LIN {X 0,Y 530.55,Z 455.718,A -85,B 0,C 180,E1 -4236.847,E2 -4236.847} C_VEL
LIN {X 0,Y 530.637,Z 451.254,A -85,B 0,C 180,E1 -4237.994,E2 -4237.994} C_VEL
LIN {X 0,Y 530.743,Z 445.924,A -85,B 0,C 180,E1 -4239.143,E2 -4239.143} C_VEL
LIN {X 0,Y 530.926,Z 439.642,A -85,B 0,C 180,E1 -4240.294,E2 -4240.294} C_VEL
LIN {X 0,Y 531.066,Z 432.27,A -85,B 0,C 180,E1 -4241.449,E2 -4241.449} C_VEL
LIN {X 0,Y 531.288,Z 425.199,A -85,B 0,C 180,E1 -4242.413,E2 -4242.413} C_VEL
LIN {X 0,Y 531.562,Z 417.094,A -85,B 0,C 180,E1 -4243.378,E2 -4243.378} C_VEL
LIN {X 0,Y 531.915,Z 406.759,A -85,B 0,C 180,E1 -4244.441,E2 -4244.441} C_VEL
LIN {X 0,Y 532.284,Z 397.021,A -85,B 0,C 180,E1 -4245.312,E2 -4245.312} C_VEL
LIN {X 0,Y 532.714,Z 385.569,A -85,B 0,C 180,E1 -4246.182,E2 -4246.182} C_VEL
LIN {X 0,Y 533.174,Z 371.646,A -85,B 0,C 180,E1 -4247.055,E2 -4247.055} C_VEL
LIN {X 0,Y 533.562,Z 358.553,A -85,B 0,C 180,E1 -4247.709,E2 -4247.709} C_VEL
LIN {X 0,Y 533.92,Z 343.815,A -85,B 0,C 180,E1 -4248.282,E2 -4248.282} C_VEL
LIN {X 0,Y 534.06,Z 328.911,A -85,B 0,C 180,E1 -4248.704,E2 -4248.704} C_VEL
LIN {X 0,Y 530.589,Z 315.52,A -85,B 0,C 180,E1 -4249.112,E2 -4249.112} C_VEL
LIN {X 0,Y 530.644,Z 311.471,A -85,B 0,C 180,E1 -4252.013,E2 -4252.013} C_VEL
LIN {X 0,Y 530.676,Z 307.059,A -85,B 0,C 180,E1 -4255.074,E2 -4255.074} C_VEL
LIN {X 0,Y 530.747,Z 303.383,A -85,B 0,C 180,E1 -4257.61,E2 -4257.61} C_VEL
LIN {X 0,Y 530.763,Z 299.76,A -85,B 0,C 180,E1 -4260.21,E2 -4260.21} C_VEL
LIN {X 0,Y 530.839,Z 296.13,A -85,B 0,C 180,E1 -4262.875,E2 -4262.875} C_VEL
LIN {X 0,Y 530.854,Z 292.306,A -85,B 0,C 180,E1 -4265.628,E2 -4265.628} C_VEL
LIN {X 0,Y 530.927,Z 287.779,A -85,B 0,C 180,E1 -4268.648,E2 -4268.648} C_VEL
LIN {X 0,Y 530.86,Z 284.993,A -85,B 0,C 180,E1 -4270.444,E2 -4270.444} C_VEL
LIN {X 0,Y 530.946,Z 284.975,A -85,B 0,C 180,E1 -4273.279,E2 -4273.279} C_VEL
LIN {X 0,Y 530.982,Z 284.971,A -85,B 0,C 180,E1 -4275.621,E2 -4275.621} C_VEL
LIN {X 0,Y 530.994,Z 284.97,A -85,B 0,C 180,E1 -4278.564,E2 -4278.564} C_VEL
LIN {X 0,Y 530.95,Z 284.971,A -85,B 0,C 180,E1 -4281.529,E2 -4281.529} C_VEL
LIN {X 0,Y 530.959,Z 284.97,A -85,B 0,C 180,E1 -4284.38,E2 -4284.38} C_VEL
LIN {X 0,Y 530.968,Z 284.973,A -85,B 0,C 180,E1 -4287.133,E2 -4287.133} C_VEL
LIN {X 0,Y 530.95,Z 284.97,A -85,B 0,C 180,E1 -4289.802,E2 -4289.802} C_VEL
LIN {X 0,Y 530.954,Z 284.97,A -85,B 0,C 180,E1 -4292.48,E2 -4292.48} C_VEL
LIN {X 0,Y 530.979,Z 284.967,A -85,B 0,C 180,E1 -4294.941,E2 -4294.941} C_VEL
LIN {X 0,Y 530.978,Z 284.964,A -85,B 0,C 180,E1 -4297.898,E2 -4297.898} C_VEL
LIN {X 0,Y 530.98,Z 284.968,A -85,B 0,C 180,E1 -4300.677,E2 -4300.677} C_VEL
LIN {X 0,Y 530.954,Z 284.967,A -85,B 0,C 180,E1 -4303.07,E2 -4303.07} C_VEL
LIN {X 0,Y 531.042,Z 284.963,A -85,B 0,C 180,E1 -4305.436,E2 -4305.436} C_VEL
LIN {X 0,Y 531.038,Z 284.96,A -85,B 0,C 180,E1 -4308.55,E2 -4308.55} C_VEL
LIN {X 0,Y 531.03,Z 284.963,A -85,B 0,C 180,E1 -4311.629,E2 -4311.629} C_VEL
LIN {X 0,Y 531.104,Z 284.947,A -85,B 0,C 180,E1 -4314.685,E2 -4314.685} C_VEL
LIN {X 0,Y 531.137,Z 284.946,A -85,B 0,C 180,E1 -4317.725,E2 -4317.725} C_VEL
LIN {X 0,Y 531.151,Z 284.945,A -85,B 0,C 180,E1 -4320.758,E2 -4320.758} C_VEL
LIN {X 0,Y 531.093,Z 284.953,A -85,B 0,C 180,E1 -4323.034,E2 -4323.034} C_VEL
LIN {X 0,Y 531.048,Z 284.955,A -85,B 0,C 180,E1 -4326.077,E2 -4326.077} C_VEL
LIN {X 0,Y 531.026,Z 284.96,A -85,B 0,C 180,E1 -4329.138,E2 -4329.138} C_VEL
LIN {X 0,Y 531.05,Z 284.956,A -85,B 0,C 180,E1 -4331.671,E2 -4331.671} C_VEL
LIN {X 0,Y 531.018,Z 284.965,A -85,B 0,C 180,E1 -4334.95,E2 -4334.95} C_VEL
LIN {X 0,Y 530.981,Z 284.965,A -85,B 0,C 180,E1 -4337.723,E2 -4337.723} C_VEL
LIN {X 0,Y 531.025,Z 284.966,A -85,B 0,C 180,E1 -4340.127,E2 -4340.127} C_VEL
LIN {X 0,Y 530.944,Z 284.97,A -85,B 0,C 180,E1 -4342.573,E2 -4342.573} C_VEL
LIN {X 0,Y 530.952,Z 284.975,A -85,B 0,C 180,E1 -4345.06,E2 -4345.06} C_VEL
LIN {X 0,Y 530.965,Z 284.968,A -85,B 0,C 180,E1 -4347.598,E2 -4347.598} C_VEL
LIN {X 0,Y 530.969,Z 284.974,A -85,B 0,C 180,E1 -4350.197,E2 -4350.197} C_VEL
LIN {X 0,Y 530.967,Z 284.968,A -85,B 0,C 180,E1 -4352.867,E2 -4352.867} C_VEL
LIN {X 0,Y 530.949,Z 284.973,A -85,B 0,C 180,E1 -4355.62,E2 -4355.62} C_VEL
LIN {X 0,Y 530.96,Z 284.975,A -85,B 0,C 180,E1 -4358.653,E2 -4358.653} C_VEL
LIN {X 0,Y 530.996,Z 284.966,A -85,B 0,C 180,E1 -4361.435,E2 -4361.435} C_VEL
LIN {X 0,Y 530.973,Z 284.966,A -85,B 0,C 180,E1 -4364.548,E2 -4364.548} C_VEL
LIN {X 0,Y 530.936,Z 284.971,A -85,B 0,C 180,E1 -4367.539,E2 -4367.539} C_VEL
LIN {X 0,Y 530.985,Z 284.972,A -85,B 0,C 180,E1 -4370.557,E2 -4370.557} C_VEL
LIN {X 0,Y 530.995,Z 285.169,A -85,B 0,C 180,E1 -4371.775,E2 -4371.775} C_VEL
LIN {X 0,Y 534.106,Z 297.132,A -85,B 0,C 180,E1 -4374.391,E2 -4374.391} C_VEL
LIN {X 0,Y 534.99,Z 301.976,A -85,B 0,C 180,E1 -4375.378,E2 -4375.378} C_VEL
LIN {X 0,Y 534.26,Z 316.689,A -85,B 0,C 180,E1 -4378.03,E2 -4378.03} C_VEL
LIN {X 0,Y 533.53,Z 334.161,A -85,B 0,C 180,E1 -4381.047,E2 -4381.047} C_VEL
LIN {X 0,Y 532.887,Z 353.224,A -85,B 0,C 180,E1 -4384.201,E2 -4384.201} C_VEL
LIN {X 0,Y 532.44,Z 368.615,A -85,B 0,C 180,E1 -4386.673,E2 -4386.673} C_VEL
LIN {X 0,Y 532.082,Z 388.428,A -85,B 0,C 180,E1 -4389.685,E2 -4389.685} C_VEL
LIN {X 0,Y 531.887,Z 396.61,A -85,B 0,C 180,E1 -4390.918,E2 -4390.918} C_VEL
LIN {X 0,Y 534.269,Z 408.735,A -85,B 0,C 180,E1 -4391.169,E2 -4391.169} C_VEL
LIN {X 0,Y 534.009,Z 424.767,A -85,B 0,C 180,E1 -4391.513,E2 -4391.513} C_VEL
LIN {X 0,Y 533.779,Z 438.733,A -85,B 0,C 180,E1 -4391.96,E2 -4391.96} C_VEL
LIN {X 0,Y 533.397,Z 452.811,A -85,B 0,C 180,E1 -4392.557,E2 -4392.557} C_VEL
LIN {X 0,Y 532.951,Z 467.093,A -85,B 0,C 180,E1 -4393.333,E2 -4393.333} C_VEL
LIN {X 0,Y 532.558,Z 480.044,A -85,B 0,C 180,E1 -4394.203,E2 -4394.203} C_VEL
LIN {X 0,Y 532.085,Z 492.083,A -85,B 0,C 180,E1 -4395.172,E2 -4395.172} C_VEL
LIN {X 0,Y 531.711,Z 503.187,A -85,B 0,C 180,E1 -4396.236,E2 -4396.236} C_VEL
LIN {X 0,Y 531.382,Z 513.39,A -85,B 0,C 180,E1 -4397.395,E2 -4397.395} C_VEL
LIN {X 0,Y 531.076,Z 523.366,A -85,B 0,C 180,E1 -4398.744,E2 -4398.744} C_VEL
LIN {X 0,Y 530.809,Z 531.647,A -85,B 0,C 180,E1 -4400.089,E2 -4400.089} C_VEL
LIN {X 0,Y 530.665,Z 539.422,A -85,B 0,C 180,E1 -4401.623,E2 -4401.623} C_VEL
LIN {X 0,Y 530.549,Z 545.605,A -85,B 0,C 180,E1 -4403.153,E2 -4403.153} C_VEL
LIN {X 0,Y 530.509,Z 550.385,A -85,B 0,C 180,E1 -4404.679,E2 -4404.679} C_VEL
LIN {X 0,Y 530.48,Z 553.887,A -85,B 0,C 180,E1 -4406.202,E2 -4406.202} C_VEL
LIN {X 0,Y 530.409,Z 556.19,A -85,B 0,C 180,E1 -4407.722,E2 -4407.722} C_VEL
LIN {X 0,Y 530.342,Z 557.348,A -85,B 0,C 180,E1 -4409.241,E2 -4409.241} C_VEL
LIN {X 0,Y 530.342,Z 557.347,A -85,B 0,C 180,E1 -4410.759,E2 -4410.759} C_VEL
LIN {X 0,Y 530.409,Z 556.186,A -85,B 0,C 180,E1 -4412.278,E2 -4412.278} C_VEL
LIN {X 0,Y 530.48,Z 553.883,A -85,B 0,C 180,E1 -4413.798,E2 -4413.798} C_VEL
LIN {X 0,Y 530.509,Z 550.386,A -85,B 0,C 180,E1 -4415.321,E2 -4415.321} C_VEL
LIN {X 0,Y 530.569,Z 545.608,A -85,B 0,C 180,E1 -4416.847,E2 -4416.847} C_VEL
LIN {X 0,Y 530.665,Z 539.419,A -85,B 0,C 180,E1 -4418.377,E2 -4418.377} C_VEL
LIN {X 0,Y 530.809,Z 531.642,A -85,B 0,C 180,E1 -4419.911,E2 -4419.911} C_VEL
LIN {X 0,Y 531.057,Z 523.365,A -85,B 0,C 180,E1 -4421.257,E2 -4421.257} C_VEL
LIN {X 0,Y 531.383,Z 513.389,A -85,B 0,C 180,E1 -4422.605,E2 -4422.605} C_VEL
LIN {X 0,Y 531.707,Z 503.182,A -85,B 0,C 180,E1 -4423.764,E2 -4423.764} C_VEL
LIN {X 0,Y 532.122,Z 491.015,A -85,B 0,C 180,E1 -4424.925,E2 -4424.925} C_VEL
LIN {X 0,Y 532.606,Z 477.588,A -85,B 0,C 180,E1 -4425.981,E2 -4425.981} C_VEL
LIN {X 0,Y 533.053,Z 463.877,A -85,B 0,C 180,E1 -4426.862,E2 -4426.862} C_VEL
LIN {X 0,Y 533.486,Z 449.795,A -85,B 0,C 180,E1 -4427.588,E2 -4427.588} C_VEL
LIN {X 0,Y 533.855,Z 435.031,A -85,B 0,C 180,E1 -4428.177,E2 -4428.177} C_VEL
LIN {X 0,Y 534.116,Z 419.224,A -85,B 0,C 180,E1 -4428.628,E2 -4428.628} C_VEL
LIN {X 0,Y 534.192,Z 408.185,A -85,B 0,C 180,E1 -4428.84,E2 -4428.84} C_VEL
LIN {X 0,Y 531.867,Z 396.393,A -85,B 0,C 180,E1 -4429.089,E2 -4429.089} C_VEL
LIN {X 0,Y 532.186,Z 378.709,A -85,B 0,C 180,E1 -4431.701,E2 -4431.701} C_VEL
LIN {X 0,Y 532.455,Z 360.86,A -85,B 0,C 180,E1 -4434.391,E2 -4434.391} C_VEL
LIN {X 0,Y 532.896,Z 342.799,A -85,B 0,C 180,E1 -4437.277,E2 -4437.277} C_VEL
LIN {X 0,Y 533.439,Z 328.196,A -85,B 0,C 180,E1 -4439.757,E2 -4439.757} C_VEL
LIN {X 0,Y 534.204,Z 314.988,A -85,B 0,C 180,E1 -4442.196,E2 -4442.196} C_VEL
LIN {X 0,Y 535.26,Z 304.386,A -85,B 0,C 180,E1 -4444.374,E2 -4444.374} C_VEL
LIN {X 0,Y 535.354,Z 302.437,A -85,B 0,C 180,E1 -4444.824,E2 -4444.824} C_VEL
LIN {X 0,Y 534.178,Z 297.091,A -85,B 0,C 180,E1 -4446.303,E2 -4446.303} C_VEL
LIN {X 0,Y 532.522,Z 291.051,A -85,B 0,C 180,E1 -4448.337,E2 -4448.337} C_VEL
LIN {X 0,Y 531.356,Z 286.461,A -85,B 0,C 180,E1 -4450.399,E2 -4450.399} C_VEL
LIN {X 0,Y 530.995,Z 284.97,A -85,B 0,C 180,E1 -4451.436,E2 -4451.436} C_VEL
LIN {X 0,Y 530.977,Z 284.972,A -85,B 0,C 180,E1 -4454.548,E2 -4454.548} C_VEL
LIN {X 0,Y 530.984,Z 284.972,A -85,B 0,C 180,E1 -4457.835,E2 -4457.835} C_VEL
LIN {X 0,Y 530.988,Z 284.972,A -85,B 0,C 180,E1 -4460.557,E2 -4460.557} C_VEL
LIN {X 0,Y 530.971,Z 285.061,A -85,B 0,C 180,E1 -4461.531,E2 -4461.531} C_VEL
LIN {X 0,Y 531.272,Z 287.127,A -85,B 0,C 180,E1 -4463.799,E2 -4463.799} C_VEL
LIN {X 0,Y 531.314,Z 289.649,A -85,B 0,C 180,E1 -4466.444,E2 -4466.444} C_VEL
LIN {X 0,Y 531.2,Z 292.331,A -85,B 0,C 180,E1 -4469.315,E2 -4469.315} C_VEL
LIN {X 0,Y 531.176,Z 294.318,A -85,B 0,C 180,E1 -4471.555,E2 -4471.555} C_VEL
LIN {X 0,Y 531.084,Z 296.552,A -85,B 0,C 180,E1 -4474.141,E2 -4474.141} C_VEL
LIN {X 0,Y 531.024,Z 298.621,A -85,B 0,C 180,E1 -4476.607,E2 -4476.607} C_VEL
LIN {X 0,Y 530.911,Z 300.717,A -85,B 0,C 180,E1 -4479.058,E2 -4479.058} C_VEL
LIN {X 0,Y 530.804,Z 302.778,A -85,B 0,C 180,E1 -4481.472,E2 -4481.472} C_VEL
LIN {X 0,Y 530.716,Z 305.487,A -85,B 0,C 180,E1 -4484.642,E2 -4484.642} C_VEL
LIN {X 0,Y 530.715,Z 307.333,A -85,B 0,C 180,E1 -4486.503,E2 -4486.503} C_VEL
LIN {X 0,Y 532.299,Z 313.645,A -85,B 0,C 180,E1 -4486.714,E2 -4486.714} C_VEL
LIN {X 0,Y 532.545,Z 319.854,A -85,B 0,C 180,E1 -4486.914,E2 -4486.914} C_VEL
LIN {X 0,Y 532.311,Z 332.527,A -85,B 0,C 180,E1 -4487.418,E2 -4487.418} C_VEL
LIN {X 0,Y 532.081,Z 343.539,A -85,B 0,C 180,E1 -4488.002,E2 -4488.002} C_VEL
LIN {X 0,Y 531.772,Z 354.747,A -85,B 0,C 180,E1 -4488.759,E2 -4488.759} C_VEL
LIN {X 0,Y 531.488,Z 365.983,A -85,B 0,C 180,E1 -4489.717,E2 -4489.717} C_VEL
LIN {X 0,Y 531.267,Z 374.976,A -85,B 0,C 180,E1 -4490.674,E2 -4490.674} C_VEL
LIN {X 0,Y 531.002,Z 383.707,A -85,B 0,C 180,E1 -4491.82,E2 -4491.82} C_VEL
LIN {X 0,Y 530.818,Z 390.721,A -85,B 0,C 180,E1 -4492.965,E2 -4492.965} C_VEL
LIN {X 0,Y 530.705,Z 397.114,A -85,B 0,C 180,E1 -4494.3,E2 -4494.3} C_VEL
LIN {X 0,Y 530.585,Z 401.337,A -85,B 0,C 180,E1 -4495.442,E2 -4495.442} C_VEL
LIN {X 0,Y 530.59,Z 403.556,A -85,B 0,C 180,E1 -4496.203,E2 -4496.203} C_VEL
LIN {X 0,Y 530.599,Z 405.354,A -85,B 0,C 180,E1 -4496.963,E2 -4496.963} C_VEL
LIN {X 0,Y 530.494,Z 406.734,A -85,B 0,C 180,E1 -4497.722,E2 -4497.722} C_VEL
LIN {X 0,Y 530.447,Z 408.296,A -85,B 0,C 180,E1 -4499.241,E2 -4499.241} C_VEL
LIN {X 0,Y 530.442,Z 408.506,A -85,B 0,C 180,E1 -4500,E2 -4500} C_VEL
LIN {X 0,Y 530.44,Z 407.737,A -85,B 0,C 180,E1 -4501.519,E2 -4501.519} C_VEL
LIN {X 0,Y 530.465,Z 406.782,A -85,B 0,C 180,E1 -4502.278,E2 -4502.278} C_VEL
LIN {X 0,Y 530.529,Z 405.422,A -85,B 0,C 180,E1 -4503.038,E2 -4503.038} C_VEL
LIN {X 0,Y 530.597,Z 402.583,A -85,B 0,C 180,E1 -4504.178,E2 -4504.178} C_VEL
LIN {X 0,Y 530.579,Z 398.752,A -85,B 0,C 180,E1 -4505.32,E2 -4505.32} C_VEL
LIN {X 0,Y 530.694,Z 394.343,A -85,B 0,C 180,E1 -4506.347,E2 -4506.347} C_VEL
LIN {X 0,Y 530.83,Z 387.534,A -85,B 0,C 180,E1 -4507.608,E2 -4507.608} C_VEL
LIN {X 0,Y 531.029,Z 379.707,A -85,B 0,C 180,E1 -4508.754,E2 -4508.754} C_VEL
LIN {X 0,Y 531.211,Z 371.719,A -85,B 0,C 180,E1 -4509.711,E2 -4509.711} C_VEL
LIN {X 0,Y 531.514,Z 361.947,A -85,B 0,C 180,E1 -4510.668,E2 -4510.668} C_VEL
LIN {X 0,Y 531.722,Z 352.361,A -85,B 0,C 180,E1 -4511.435,E2 -4511.435} C_VEL
LIN {X 0,Y 531.966,Z 340.299,A -85,B 0,C 180,E1 -4512.203,E2 -4512.203} C_VEL
LIN {X 0,Y 532.221,Z 327.432,A -85,B 0,C 180,E1 -4512.827,E2 -4512.827} C_VEL
LIN {X 0,Y 532.318,Z 314.68,A -85,B 0,C 180,E1 -4513.274,E2 -4513.274} C_VEL
LIN {X 0,Y 530.496,Z 305.726,A -85,B 0,C 180,E1 -4513.552,E2 -4513.552} C_VEL
LIN {X 0,Y 530.505,Z 303.016,A -85,B 0,C 180,E1 -4516.153,E2 -4516.153} C_VEL
LIN {X 0,Y 530.558,Z 299.64,A -85,B 0,C 180,E1 -4519.339,E2 -4519.339} C_VEL
LIN {X 0,Y 530.568,Z 296.85,A -85,B 0,C 180,E1 -4521.992,E2 -4521.992} C_VEL
LIN {X 0,Y 530.609,Z 293.542,A -85,B 0,C 180,E1 -4525.078,E2 -4525.078} C_VEL
LIN {X 0,Y 530.658,Z 290.857,A -85,B 0,C 180,E1 -4527.616,E2 -4527.616} C_VEL
LIN {X 0,Y 530.662,Z 288.005,A -85,B 0,C 180,E1 -4530.216,E2 -4530.216} C_VEL
LIN {X 0,Y 530.626,Z 285.135,A -85,B 0,C 180,E1 -4532.891,E2 -4532.891} C_VEL
LIN {X 0,Y 530.907,Z 284.979,A -85,B 0,C 180,E1 -4535.624,E2 -4535.624} C_VEL
LIN {X 0,Y 530.963,Z 284.969,A -85,B 0,C 180,E1 -4538.47,E2 -4538.47} C_VEL
LIN {X 0,Y 530.985,Z 284.965,A -85,B 0,C 180,E1 -4539.611,E2 -4539.611} C_VEL
LIN {X 0,Y 530.311,Z 285.051,A -85,B 0,C 180,E1 -4540.244,E2 -4540.244} C_VEL
LIN {X 0,Y 527.447,Z 285.406,A -85,B 0,C 180,E1 -4541.271,E2 -4541.271} C_VEL
LIN {X 0,Y 525.032,Z 285.708,A -85,B 0,C 180,E1 -4542.099,E2 -4542.099} C_VEL
LIN {X 0,Y 523.998,Z 285.839,A -85,B 0,C 180,E1 -4542.737,E2 -4542.737} C_VEL
LIN {X 0,Y 523.916,Z 285.845,A -85,B 0,C 180,E1 -4542.954,E2 -4542.954} C_VEL
LIN {X 0,Y 523.927,Z 285.847,A -85,B 0,C 180,E1 -4545.77,E2 -4545.77} C_VEL
LIN {X 0,Y 523.856,Z 285.856,A -85,B 0,C 180,E1 -4548.899,E2 -4548.899} C_VEL
LIN {X 0,Y 523.853,Z 286.229,A -85,B 0,C 180,E1 -4549.911,E2 -4549.911} C_VEL
LIN {X 0,Y 523.84,Z 290.026,A -85,B 0,C 180,E1 -4552.332,E2 -4552.332} C_VEL
LIN {X 0,Y 523.793,Z 293.791,A -85,B 0,C 180,E1 -4554.932,E2 -4554.932} C_VEL
LIN {X 0,Y 523.797,Z 297.608,A -85,B 0,C 180,E1 -4557.704,E2 -4557.704} C_VEL
LIN {X 0,Y 523.704,Z 301.712,A -85,B 0,C 180,E1 -4560.726,E2 -4560.726} C_VEL
LIN {X 0,Y 523.656,Z 306.399,A -85,B 0,C 180,E1 -4564.054,E2 -4564.054} C_VEL
LIN {X 0,Y 523.605,Z 310.847,A -85,B 0,C 180,E1 -4567.092,E2 -4567.092} C_VEL
LIN {X 0,Y 523.587,Z 315.58,A -85,B 0,C 180,E1 -4570.393,E2 -4570.393} C_VEL
LIN {X 0,Y 523.564,Z 316.054,A -85,B 0,C 180,E1 -4570.728,E2 -4570.728} C_VEL
LIN {X 0,Y 527.46,Z 330.475,A -85,B 0,C 180,E1 -4571.169,E2 -4571.169} C_VEL
LIN {X 0,Y 527.204,Z 345.774,A -85,B 0,C 180,E1 -4571.617,E2 -4571.617} C_VEL
LIN {X 0,Y 526.731,Z 360.928,A -85,B 0,C 180,E1 -4572.229,E2 -4572.229} C_VEL
LIN {X 0,Y 526.363,Z 374.055,A -85,B 0,C 180,E1 -4572.918,E2 -4572.918} C_VEL
LIN {X 0,Y 525.834,Z 387.661,A -85,B 0,C 180,E1 -4573.799,E2 -4573.799} C_VEL
LIN {X 0,Y 525.366,Z 400.033,A -85,B 0,C 180,E1 -4574.78,E2 -4574.78} C_VEL
LIN {X 0,Y 524.902,Z 411.392,A -85,B 0,C 180,E1 -4575.856,E2 -4575.856} C_VEL
LIN {X 0,Y 524.499,Z 421.791,A -85,B 0,C 180,E1 -4577.03,E2 -4577.03} C_VEL
LIN {X 0,Y 524.096,Z 430.656,A -85,B 0,C 180,E1 -4578.213,E2 -4578.213} C_VEL
LIN {X 0,Y 523.963,Z 438.024,A -85,B 0,C 180,E1 -4579.372,E2 -4579.372} C_VEL
LIN {X 0,Y 523.701,Z 445.451,A -85,B 0,C 180,E1 -4580.733,E2 -4580.733} C_VEL
LIN {X 0,Y 523.536,Z 452.535,A -85,B 0,C 180,E1 -4582.285,E2 -4582.285} C_VEL
LIN {X 0,Y 523.423,Z 458.003,A -85,B 0,C 180,E1 -4583.833,E2 -4583.833} C_VEL
LIN {X 0,Y 523.441,Z 460.258,A -85,B 0,C 180,E1 -4584.607,E2 -4584.607} C_VEL
LIN {X 0,Y 523.402,Z 463.836,A -85,B 0,C 180,E1 -4586.15,E2 -4586.15} C_VEL
LIN {X 0,Y 523.333,Z 466.123,A -85,B 0,C 180,E1 -4587.691,E2 -4587.691} C_VEL
LIN {X 0,Y 523.246,Z 467.265,A -85,B 0,C 180,E1 -4589.23,E2 -4589.23} C_VEL
LIN {X 0,Y 523.244,Z 467.497,A -85,B 0,C 180,E1 -4590,E2 -4590} C_VEL
LIN {X 0,Y 523.273,Z 466.938,A -85,B 0,C 180,E1 -4591.539,E2 -4591.539} C_VEL
LIN {X 0,Y 523.359,Z 465.219,A -85,B 0,C 180,E1 -4593.079,E2 -4593.079} C_VEL
LIN {X 0,Y 523.402,Z 463.995,A -85,B 0,C 180,E1 -4593.849,E2 -4593.849} C_VEL
LIN {X 0,Y 523.44,Z 460.522,A -85,B 0,C 180,E1 -4595.393,E2 -4595.393} C_VEL
LIN {X 0,Y 523.481,Z 455.711,A -85,B 0,C 180,E1 -4596.94,E2 -4596.94} C_VEL
LIN {X 0,Y 523.562,Z 451.244,A -85,B 0,C 180,E1 -4598.102,E2 -4598.102} C_VEL
LIN {X 0,Y 523.666,Z 445.915,A -85,B 0,C 180,E1 -4599.268,E2 -4599.268} C_VEL
LIN {X 0,Y 523.952,Z 438.549,A -85,B 0,C 180,E1 -4600.628,E2 -4600.628} C_VEL
LIN {X 0,Y 524.086,Z 431.295,A -85,B 0,C 180,E1 -4601.782,E2 -4601.782} C_VEL
LIN {X 0,Y 524.477,Z 422.512,A -85,B 0,C 180,E1 -4602.97,E2 -4602.97} C_VEL
LIN {X 0,Y 524.883,Z 412.256,A -85,B 0,C 180,E1 -4604.144,E2 -4604.144} C_VEL
LIN {X 0,Y 525.386,Z 400.02,A -85,B 0,C 180,E1 -4605.312,E2 -4605.312} C_VEL
LIN {X 0,Y 525.86,Z 387.531,A -85,B 0,C 180,E1 -4606.299,E2 -4606.299} C_VEL
LIN {X 0,Y 526.375,Z 373.882,A -85,B 0,C 180,E1 -4607.182,E2 -4607.182} C_VEL
LIN {X 0,Y 526.771,Z 360.713,A -85,B 0,C 180,E1 -4607.87,E2 -4607.87} C_VEL
LIN {X 0,Y 527.188,Z 345.994,A -85,B 0,C 180,E1 -4608.466,E2 -4608.466} C_VEL
LIN {X 0,Y 527.476,Z 330.668,A -85,B 0,C 180,E1 -4608.916,E2 -4608.916} C_VEL
LIN {X 0,Y 524.21,Z 318.376,A -85,B 0,C 180,E1 -4609.296,E2 -4609.296} C_VEL
LIN {X 0,Y 523.576,Z 316.052,A -85,B 0,C 180,E1 -4609.378,E2 -4609.378} C_VEL
LIN {X 0,Y 523.599,Z 312.078,A -85,B 0,C 180,E1 -4612.157,E2 -4612.157} C_VEL
LIN {X 0,Y 523.619,Z 308.498,A -85,B 0,C 180,E1 -4614.587,E2 -4614.587} C_VEL
LIN {X 0,Y 523.653,Z 304.79,A -85,B 0,C 180,E1 -4617.15,E2 -4617.15} C_VEL
LIN {X 0,Y 523.708,Z 301.169,A -85,B 0,C 180,E1 -4619.77,E2 -4619.77} C_VEL
LIN {X 0,Y 523.795,Z 297.529,A -85,B 0,C 180,E1 -4622.459,E2 -4622.459} C_VEL
LIN {X 0,Y 523.792,Z 293.7,A -85,B 0,C 180,E1 -4625.236,E2 -4625.236} C_VEL
LIN {X 0,Y 523.87,Z 289.504,A -85,B 0,C 180,E1 -4628.106,E2 -4628.106} C_VEL
LIN {X 0,Y 523.834,Z 286.321,A -85,B 0,C 180,E1 -4630.116,E2 -4630.116} C_VEL
LIN {X 0,Y 523.882,Z 285.859,A -85,B 0,C 180,E1 -4631.301,E2 -4631.301} C_VEL
LIN {X 0,Y 523.934,Z 285.847,A -85,B 0,C 180,E1 -4634.229,E2 -4634.229} C_VEL
LIN {X 0,Y 523.917,Z 285.853,A -85,B 0,C 180,E1 -4636.833,E2 -4636.833} C_VEL
LIN {X 0,Y 523.939,Z 285.847,A -85,B 0,C 180,E1 -4638.908,E2 -4638.908} C_VEL
LIN {X 0,Y 523.911,Z 285.852,A -85,B 0,C 180,E1 -4641.898,E2 -4641.898} C_VEL
LIN {X 0,Y 523.932,Z 285.847,A -85,B 0,C 180,E1 -4644.91,E2 -4644.91} C_VEL
LIN {X 0,Y 523.936,Z 285.845,A -85,B 0,C 180,E1 -4647.68,E2 -4647.68} C_VEL
LIN {X 0,Y 523.935,Z 285.846,A -85,B 0,C 180,E1 -4650.68,E2 -4650.68} C_VEL
LIN {X 0,Y 523.907,Z 285.849,A -85,B 0,C 180,E1 -4653.725,E2 -4653.725} C_VEL
LIN {X 0,Y 523.913,Z 285.848,A -85,B 0,C 180,E1 -4656.27,E2 -4656.27} C_VEL
LIN {X 0,Y 523.946,Z 285.845,A -85,B 0,C 180,E1 -4658.767,E2 -4658.767} C_VEL
LIN {X 0,Y 523.934,Z 285.845,A -85,B 0,C 180,E1 -4661.22,E2 -4661.22} C_VEL
LIN {X 0,Y 523.905,Z 285.849,A -85,B 0,C 180,E1 -4663.638,E2 -4663.638} C_VEL
LIN {X 0,Y 523.946,Z 285.843,A -85,B 0,C 180,E1 -4666.028,E2 -4666.028} C_VEL
LIN {X 0,Y 524.014,Z 285.834,A -85,B 0,C 180,E1 -4668.394,E2 -4668.394} C_VEL
LIN {X 0,Y 523.983,Z 285.84,A -85,B 0,C 180,E1 -4671.516,E2 -4671.516} C_VEL
LIN {X 0,Y 524.064,Z 285.824,A -85,B 0,C 180,E1 -4674.613,E2 -4674.613} C_VEL
LIN {X 0,Y 524.11,Z 285.822,A -85,B 0,C 180,E1 -4677.694,E2 -4677.694} C_VEL
LIN {X 0,Y 524.122,Z 285.82,A -85,B 0,C 180,E1 -4680.768,E2 -4680.768} C_VEL
LIN {X 0,Y 524.034,Z 285.833,A -85,B 0,C 180,E1 -4683.075,E2 -4683.075} C_VEL
LIN {X 0,Y 524.014,Z 285.831,A -85,B 0,C 180,E1 -4686.159,E2 -4686.159} C_VEL
LIN {X 0,Y 523.996,Z 285.836,A -85,B 0,C 180,E1 -4689.262,E2 -4689.262} C_VEL
LIN {X 0,Y 524,Z 285.834,A -85,B 0,C 180,E1 -4691.737,E2 -4691.737} C_VEL
LIN {X 0,Y 523.983,Z 285.842,A -85,B 0,C 180,E1 -4695.048,E2 -4695.048} C_VEL
LIN {X 0,Y 523.948,Z 285.842,A -85,B 0,C 180,E1 -4697.969,E2 -4697.969} C_VEL
LIN {X 0,Y 523.973,Z 285.841,A -85,B 0,C 180,E1 -4700.41,E2 -4700.41} C_VEL
LIN {X 0,Y 523.909,Z 285.846,A -85,B 0,C 180,E1 -4702.894,E2 -4702.894} C_VEL
LIN {X 0,Y 523.9,Z 285.85,A -85,B 0,C 180,E1 -4705.421,E2 -4705.421} C_VEL
LIN {X 0,Y 523.915,Z 285.846,A -85,B 0,C 180,E1 -4708.002,E2 -4708.002} C_VEL
LIN {X 0,Y 523.945,Z 285.844,A -85,B 0,C 180,E1 -4710.855,E2 -4710.855} C_VEL
LIN {X 0,Y 523.959,Z 285.846,A -85,B 0,C 180,E1 -4713.734,E2 -4713.734} C_VEL
LIN {X 0,Y 523.896,Z 285.85,A -85,B 0,C 180,E1 -4716.4,E2 -4716.4} C_VEL
LIN {X 0,Y 523.911,Z 285.849,A -85,B 0,C 180,E1 -4719.086,E2 -4719.086} C_VEL
LIN {X 0,Y 523.954,Z 285.844,A -85,B 0,C 180,E1 -4722.119,E2 -4722.119} C_VEL
LIN {X 0,Y 523.942,Z 285.845,A -85,B 0,C 180,E1 -4725.31,E2 -4725.31} C_VEL
LIN {X 0,Y 523.922,Z 285.849,A -85,B 0,C 180,E1 -4728.694,E2 -4728.694} C_VEL
LIN {X 0,Y 523.959,Z 285.974,A -85,B 0,C 180,E1 -4731.33,E2 -4731.33} C_VEL
LIN {X 0,Y 527.118,Z 298.309,A -85,B 0,C 180,E1 -4734.081,E2 -4734.081} C_VEL
LIN {X 0,Y 528.241,Z 303.141,A -85,B 0,C 180,E1 -4735.104,E2 -4735.104} C_VEL
LIN {X 0,Y 527.603,Z 315.476,A -85,B 0,C 180,E1 -4737.382,E2 -4737.382} C_VEL
LIN {X 0,Y 526.872,Z 330.905,A -85,B 0,C 180,E1 -4740.117,E2 -4740.117} C_VEL
LIN {X 0,Y 526.182,Z 347.775,A -85,B 0,C 180,E1 -4742.992,E2 -4742.992} C_VEL
LIN {X 0,Y 525.582,Z 366.851,A -85,B 0,C 180,E1 -4746.14,E2 -4746.14} C_VEL
LIN {X 0,Y 525.105,Z 388.156,A -85,B 0,C 180,E1 -4749.452,E2 -4749.452} C_VEL
LIN {X 0,Y 524.869,Z 396.174,A -85,B 0,C 180,E1 -4750.687,E2 -4750.687} C_VEL
LIN {X 0,Y 527.418,Z 410.234,A -85,B 0,C 180,E1 -4750.986,E2 -4750.986} C_VEL
LIN {X 0,Y 527.161,Z 426.299,A -85,B 0,C 180,E1 -4751.36,E2 -4751.36} C_VEL
LIN {X 0,Y 526.829,Z 441.078,A -85,B 0,C 180,E1 -4751.862,E2 -4751.862} C_VEL
LIN {X 0,Y 526.396,Z 455.751,A -85,B 0,C 180,E1 -4752.518,E2 -4752.518} C_VEL
LIN {X 0,Y 525.937,Z 469.641,A -85,B 0,C 180,E1 -4753.304,E2 -4753.304} C_VEL
LIN {X 0,Y 525.5,Z 483.767,A -85,B 0,C 180,E1 -4754.287,E2 -4754.287} C_VEL
LIN {X 0,Y 525.057,Z 495.281,A -85,B 0,C 180,E1 -4755.267,E2 -4755.267} C_VEL
LIN {X 0,Y 524.625,Z 506.746,A -85,B 0,C 180,E1 -4756.442,E2 -4756.442} C_VEL
LIN {X 0,Y 524.293,Z 516.389,A -85,B 0,C 180,E1 -4757.615,E2 -4757.615} C_VEL
LIN {X 0,Y 524.032,Z 525.854,A -85,B 0,C 180,E1 -4758.982,E2 -4758.982} C_VEL
LIN {X 0,Y 523.697,Z 533.736,A -85,B 0,C 180,E1 -4760.343,E2 -4760.343} C_VEL
LIN {X 0,Y 523.564,Z 541.091,A -85,B 0,C 180,E1 -4761.898,E2 -4761.898} C_VEL
LIN {X 0,Y 523.468,Z 546.993,A -85,B 0,C 180,E1 -4763.469,E2 -4763.469} C_VEL
LIN {X 0,Y 523.442,Z 550.385,A -85,B 0,C 180,E1 -4764.607,E2 -4764.607} C_VEL
LIN {X 0,Y 523.401,Z 553.887,A -85,B 0,C 180,E1 -4766.151,E2 -4766.151} C_VEL
LIN {X 0,Y 523.332,Z 556.19,A -85,B 0,C 180,E1 -4767.691,E2 -4767.691} C_VEL
LIN {X 0,Y 523.248,Z 557.348,A -85,B 0,C 180,E1 -4769.231,E2 -4769.231} C_VEL
LIN {X 0,Y 523.248,Z 557.347,A -85,B 0,C 180,E1 -4770.77,E2 -4770.77} C_VEL
LIN {X 0,Y 523.332,Z 556.185,A -85,B 0,C 180,E1 -4772.309,E2 -4772.309} C_VEL
LIN {X 0,Y 523.401,Z 553.882,A -85,B 0,C 180,E1 -4773.85,E2 -4773.85} C_VEL
LIN {X 0,Y 523.442,Z 550.386,A -85,B 0,C 180,E1 -4775.393,E2 -4775.393} C_VEL
LIN {X 0,Y 523.49,Z 545.609,A -85,B 0,C 180,E1 -4776.94,E2 -4776.94} C_VEL
LIN {X 0,Y 523.612,Z 539.419,A -85,B 0,C 180,E1 -4778.491,E2 -4778.491} C_VEL
LIN {X 0,Y 523.776,Z 531.641,A -85,B 0,C 180,E1 -4780.046,E2 -4780.046} C_VEL
LIN {X 0,Y 524.019,Z 523.365,A -85,B 0,C 180,E1 -4781.41,E2 -4781.41} C_VEL
LIN {X 0,Y 524.381,Z 513.389,A -85,B 0,C 180,E1 -4782.776,E2 -4782.776} C_VEL
LIN {X 0,Y 524.76,Z 503.181,A -85,B 0,C 180,E1 -4783.95,E2 -4783.95} C_VEL
LIN {X 0,Y 525.167,Z 492.054,A -85,B 0,C 180,E1 -4785.028,E2 -4785.028} C_VEL
LIN {X 0,Y 525.656,Z 479.788,A -85,B 0,C 180,E1 -4786.007,E2 -4786.007} C_VEL
LIN {X 0,Y 526.053,Z 466.262,A -85,B 0,C 180,E1 -4786.893,E2 -4786.893} C_VEL
LIN {X 0,Y 526.466,Z 452.419,A -85,B 0,C 180,E1 -4787.63,E2 -4787.63} C_VEL
LIN {X 0,Y 526.876,Z 438.269,A -85,B 0,C 180,E1 -4788.227,E2 -4788.227} C_VEL
LIN {X 0,Y 527.139,Z 423.178,A -85,B 0,C 180,E1 -4788.707,E2 -4788.707} C_VEL
LIN {X 0,Y 527.306,Z 409.059,A -85,B 0,C 180,E1 -4789.02,E2 -4789.02} C_VEL
LIN {X 0,Y 524.802,Z 395.692,A -85,B 0,C 180,E1 -4789.308,E2 -4789.308} C_VEL
LIN {X 0,Y 525.16,Z 379.105,A -85,B 0,C 180,E1 -4791.8,E2 -4791.8} C_VEL
LIN {X 0,Y 525.444,Z 362.898,A -85,B 0,C 180,E1 -4794.286,E2 -4794.286} C_VEL
LIN {X 0,Y 525.929,Z 344.715,A -85,B 0,C 180,E1 -4797.238,E2 -4797.238} C_VEL
LIN {X 0,Y 526.558,Z 329.794,A -85,B 0,C 180,E1 -4799.824,E2 -4799.824} C_VEL
LIN {X 0,Y 527.376,Z 317.207,A -85,B 0,C 180,E1 -4802.212,E2 -4802.212} C_VEL
LIN {X 0,Y 528.538,Z 306.47,A -85,B 0,C 180,E1 -4804.471,E2 -4804.471} C_VEL
LIN {X 0,Y 528.409,Z 303.161,A -85,B 0,C 180,E1 -4805.286,E2 -4805.286} C_VEL
LIN {X 0,Y 527.074,Z 297.852,A -85,B 0,C 180,E1 -4806.872,E2 -4806.872} C_VEL
LIN {X 0,Y 525.466,Z 291.772,A -85,B 0,C 180,E1 -4809.128,E2 -4809.128} C_VEL
LIN {X 0,Y 524.47,Z 288.039,A -85,B 0,C 180,E1 -4811.042,E2 -4811.042} C_VEL
LIN {X 0,Y 523.94,Z 285.848,A -85,B 0,C 180,E1 -4812.779,E2 -4812.779} C_VEL
LIN {X 0,Y 523.932,Z 285.85,A -85,B 0,C 180,E1 -4815.771,E2 -4815.771} C_VEL
LIN {X 0,Y 523.941,Z 285.849,A -85,B 0,C 180,E1 -4818.908,E2 -4818.908} C_VEL
LIN {X 0,Y 523.951,Z 285.848,A -85,B 0,C 180,E1 -4819.921,E2 -4819.921} C_VEL
LIN {X 0,Y 524.173,Z 287.363,A -85,B 0,C 180,E1 -4822.285,E2 -4822.285} C_VEL
LIN {X 0,Y 524.35,Z 289.585,A -85,B 0,C 180,E1 -4824.846,E2 -4824.846} C_VEL
LIN {X 0,Y 524.307,Z 292.104,A -85,B 0,C 180,E1 -4827.616,E2 -4827.616} C_VEL
LIN {X 0,Y 524.209,Z 294.767,A -85,B 0,C 180,E1 -4830.628,E2 -4830.628} C_VEL
LIN {X 0,Y 524.11,Z 297.402,A -85,B 0,C 180,E1 -4833.736,E2 -4833.736} C_VEL
LIN {X 0,Y 524.025,Z 299.537,A -85,B 0,C 180,E1 -4836.275,E2 -4836.275} C_VEL
LIN {X 0,Y 523.918,Z 301.635,A -85,B 0,C 180,E1 -4838.766,E2 -4838.766} C_VEL
LIN {X 0,Y 523.814,Z 303.733,A -85,B 0,C 180,E1 -4841.216,E2 -4841.216} C_VEL
LIN {X 0,Y 523.759,Z 305.83,A -85,B 0,C 180,E1 -4843.633,E2 -4843.633} C_VEL
LIN {X 0,Y 523.673,Z 308.192,A -85,B 0,C 180,E1 -4846.281,E2 -4846.281} C_VEL
LIN {X 0,Y 525.462,Z 314.341,A -85,B 0,C 180,E1 -4846.501,E2 -4846.501} C_VEL
LIN {X 0,Y 525.765,Z 320.158,A -85,B 0,C 180,E1 -4846.693,E2 -4846.693} C_VEL
LIN {X 0,Y 525.521,Z 332.491,A -85,B 0,C 180,E1 -4847.183,E2 -4847.183} C_VEL
LIN {X 0,Y 525.263,Z 344.197,A -85,B 0,C 180,E1 -4847.804,E2 -4847.804} C_VEL
LIN {X 0,Y 524.91,Z 355.959,A -85,B 0,C 180,E1 -4848.61,E2 -4848.61} C_VEL
LIN {X 0,Y 524.597,Z 367.154,A -85,B 0,C 180,E1 -4849.58,E2 -4849.58} C_VEL
LIN {X 0,Y 524.366,Z 376.116,A -85,B 0,C 180,E1 -4850.55,E2 -4850.55} C_VEL
LIN {X 0,Y 524.07,Z 384.827,A -85,B 0,C 180,E1 -4851.711,E2 -4851.711} C_VEL
LIN {X 0,Y 523.87,Z 391.83,A -85,B 0,C 180,E1 -4852.872,E2 -4852.872} C_VEL
LIN {X 0,Y 523.806,Z 396.551,A -85,B 0,C 180,E1 -4853.838,E2 -4853.838} C_VEL
LIN {X 0,Y 523.598,Z 401.15,A -85,B 0,C 180,E1 -4854.995,E2 -4854.995} C_VEL
LIN {X 0,Y 523.589,Z 404.639,A -85,B 0,C 180,E1 -4856.152,E2 -4856.152} C_VEL
LIN {X 0,Y 523.613,Z 406.426,A -85,B 0,C 180,E1 -4856.922,E2 -4856.922} C_VEL
LIN {X 0,Y 523.497,Z 407.801,A -85,B 0,C 180,E1 -4857.692,E2 -4857.692} C_VEL
LIN {X 0,Y 523.448,Z 409.339,A -85,B 0,C 180,E1 -4859.231,E2 -4859.231} C_VEL
LIN {X 0,Y 523.44,Z 409.538,A -85,B 0,C 180,E1 -4860,E2 -4860} C_VEL
LIN {X 0,Y 523.427,Z 408.749,A -85,B 0,C 180,E1 -4861.539,E2 -4861.539} C_VEL
LIN {X 0,Y 523.506,Z 406.396,A -85,B 0,C 180,E1 -4863.078,E2 -4863.078} C_VEL
LIN {X 0,Y 523.589,Z 403.528,A -85,B 0,C 180,E1 -4864.234,E2 -4864.234} C_VEL
LIN {X 0,Y 523.574,Z 399.668,A -85,B 0,C 180,E1 -4865.392,E2 -4865.392} C_VEL
LIN {X 0,Y 523.716,Z 394.042,A -85,B 0,C 180,E1 -4866.676,E2 -4866.676} C_VEL
LIN {X 0,Y 523.879,Z 387.188,A -85,B 0,C 180,E1 -4867.904,E2 -4867.904} C_VEL
LIN {X 0,Y 524.078,Z 379.059,A -85,B 0,C 180,E1 -4869.066,E2 -4869.066} C_VEL
LIN {X 0,Y 524.304,Z 370.742,A -85,B 0,C 180,E1 -4870.036,E2 -4870.036} C_VEL
LIN {X 0,Y 524.614,Z 360.492,A -85,B 0,C 180,E1 -4871.005,E2 -4871.005} C_VEL
LIN {X 0,Y 524.856,Z 350.024,A -85,B 0,C 180,E1 -4871.807,E2 -4871.807} C_VEL
LIN {X 0,Y 525.139,Z 339.338,A -85,B 0,C 180,E1 -4872.463,E2 -4872.463} C_VEL
LIN {X 0,Y 525.377,Z 327.134,A -85,B 0,C 180,E1 -4873.046,E2 -4873.046} C_VEL
LIN {X 0,Y 525.441,Z 315.695,A -85,B 0,C 180,E1 -4873.451,E2 -4873.451} C_VEL
LIN {X 0,Y 523.443,Z 306.283,A -85,B 0,C 180,E1 -4873.763,E2 -4873.763} C_VEL
LIN {X 0,Y 523.437,Z 303.506,A -85,B 0,C 180,E1 -4876.377,E2 -4876.377} C_VEL
LIN {X 0,Y 523.507,Z 300.052,A -85,B 0,C 180,E1 -4879.61,E2 -4879.61} C_VEL
LIN {X 0,Y 523.498,Z 297.404,A -85,B 0,C 180,E1 -4882.129,E2 -4882.129} C_VEL
LIN {X 0,Y 523.544,Z 294.768,A -85,B 0,C 180,E1 -4884.591,E2 -4884.591} C_VEL
LIN {X 0,Y 523.608,Z 291.48,A -85,B 0,C 180,E1 -4887.641,E2 -4887.641} C_VEL
LIN {X 0,Y 523.584,Z 288.046,A -85,B 0,C 180,E1 -4890.788,E2 -4890.788} C_VEL
LIN {X 0,Y 523.547,Z 286.268,A -85,B 0,C 180,E1 -4892.477,E2 -4892.477} C_VEL
LIN {X 0,Y 523.766,Z 285.87,A -85,B 0,C 180,E1 -4894.303,E2 -4894.303} C_VEL
LIN {X 0,Y 523.906,Z 285.854,A -85,B 0,C 180,E1 -4897.132,E2 -4897.132} C_VEL
LIN {X 0,Y 523.941,Z 285.842,A -85,B 0,C 180,E1 -4900.13,E2 -4900.13} C_VEL
LIN {X 0,Y 523.916,Z 285.845,A -85,B 0,C 180,E1 -4902.954,E2 -4902.954} C_VEL
LIN {X 0,Y 523.26,Z 285.927,A -85,B 0,C 180,E1 -4903.595,E2 -4903.595} C_VEL
LIN {X 0,Y 520.426,Z 286.285,A -85,B 0,C 180,E1 -4904.637,E2 -4904.637} C_VEL
LIN {X 0,Y 518.013,Z 286.588,A -85,B 0,C 180,E1 -4905.476,E2 -4905.476} C_VEL
LIN {X 0,Y 516.956,Z 286.718,A -85,B 0,C 180,E1 -4906.124,E2 -4906.124} C_VEL
LIN {X 0,Y 516.86,Z 286.728,A -85,B 0,C 180,E1 -4906.344,E2 -4906.344} C_VEL
LIN {X 0,Y 516.777,Z 286.74,A -85,B 0,C 180,E1 -4909.248,E2 -4909.248} C_VEL
LIN {X 0,Y 516.77,Z 286.921,A -85,B 0,C 180,E1 -4909.774,E2 -4909.774} C_VEL
LIN {X 0,Y 516.792,Z 290.783,A -85,B 0,C 180,E1 -4912.268,E2 -4912.268} C_VEL
LIN {X 0,Y 516.763,Z 294.984,A -85,B 0,C 180,E1 -4915.166,E2 -4915.166} C_VEL
LIN {X 0,Y 516.715,Z 298.802,A -85,B 0,C 180,E1 -4917.964,E2 -4917.964} C_VEL
LIN {X 0,Y 516.665,Z 302.476,A -85,B 0,C 180,E1 -4920.679,E2 -4920.679} C_VEL
LIN {X 0,Y 516.585,Z 306.893,A -85,B 0,C 180,E1 -4923.885,E2 -4923.885} C_VEL
LIN {X 0,Y 516.533,Z 311.143,A -85,B 0,C 180,E1 -4926.76,E2 -4926.76} C_VEL
LIN {X 0,Y 516.559,Z 316.056,A -85,B 0,C 180,E1 -4930.115,E2 -4930.115} C_VEL
LIN {X 0,Y 516.565,Z 316.542,A -85,B 0,C 180,E1 -4930.45,E2 -4930.45} C_VEL
LIN {X 0,Y 520.145,Z 329.137,A -85,B 0,C 180,E1 -4930.846,E2 -4930.846} C_VEL
LIN {X 0,Y 520.785,Z 333.025,A -85,B 0,C 180,E1 -4930.967,E2 -4930.967} C_VEL
LIN {X 0,Y 520.493,Z 348.025,A -85,B 0,C 180,E1 -4931.431,E2 -4931.431} C_VEL
LIN {X 0,Y 519.991,Z 362.588,A -85,B 0,C 180,E1 -4932.041,E2 -4932.041} C_VEL
LIN {X 0,Y 519.56,Z 376.34,A -85,B 0,C 180,E1 -4932.788,E2 -4932.788} C_VEL
LIN {X 0,Y 519.018,Z 389.627,A -85,B 0,C 180,E1 -4933.682,E2 -4933.682} C_VEL
LIN {X 0,Y 518.473,Z 401.949,A -85,B 0,C 180,E1 -4934.689,E2 -4934.689} C_VEL
LIN {X 0,Y 517.961,Z 413.871,A -85,B 0,C 180,E1 -4935.863,E2 -4935.863} C_VEL
LIN {X 0,Y 517.501,Z 423.964,A -85,B 0,C 180,E1 -4937.051,E2 -4937.051} C_VEL
LIN {X 0,Y 517.102,Z 433.822,A -85,B 0,C 180,E1 -4938.435,E2 -4938.435} C_VEL
LIN {X 0,Y 516.796,Z 441.998,A -85,B 0,C 180,E1 -4939.817,E2 -4939.817} C_VEL
LIN {X 0,Y 516.578,Z 449.655,A -85,B 0,C 180,E1 -4941.393,E2 -4941.393} C_VEL
LIN {X 0,Y 516.424,Z 455.706,A -85,B 0,C 180,E1 -4942.965,E2 -4942.965} C_VEL
LIN {X 0,Y 516.373,Z 460.444,A -85,B 0,C 180,E1 -4944.533,E2 -4944.533} C_VEL
LIN {X 0,Y 516.307,Z 463.908,A -85,B 0,C 180,E1 -4946.097,E2 -4946.097} C_VEL
LIN {X 0,Y 516.259,Z 466.145,A -85,B 0,C 180,E1 -4947.659,E2 -4947.659} C_VEL
LIN {X 0,Y 516.156,Z 467.259,A -85,B 0,C 180,E1 -4949.22,E2 -4949.22} C_VEL
LIN {X 0,Y 516.152,Z 467.497,A -85,B 0,C 180,E1 -4950,E2 -4950} C_VEL
LIN {X 0,Y 516.19,Z 466.94,A -85,B 0,C 180,E1 -4951.56,E2 -4951.56} C_VEL
LIN {X 0,Y 516.273,Z 465.266,A -85,B 0,C 180,E1 -4953.121,E2 -4953.121} C_VEL
LIN {X 0,Y 516.308,Z 464.068,A -85,B 0,C 180,E1 -4953.902,E2 -4953.902} C_VEL
LIN {X 0,Y 516.386,Z 459.613,A -85,B 0,C 180,E1 -4955.858,E2 -4955.858} C_VEL
LIN {X 0,Y 516.428,Z 454.658,A -85,B 0,C 180,E1 -4957.428,E2 -4957.428} C_VEL
LIN {X 0,Y 516.607,Z 448.306,A -85,B 0,C 180,E1 -4959.001,E2 -4959.001} C_VEL
LIN {X 0,Y 516.86,Z 441.404,A -85,B 0,C 180,E1 -4960.379,E2 -4960.379} C_VEL
LIN {X 0,Y 517.113,Z 433.11,A -85,B 0,C 180,E1 -4961.763,E2 -4961.763} C_VEL
LIN {X 0,Y 517.565,Z 423.101,A -85,B 0,C 180,E1 -4963.147,E2 -4963.147} C_VEL
LIN {X 0,Y 518.024,Z 412.836,A -85,B 0,C 180,E1 -4964.335,E2 -4964.335} C_VEL
LIN {X 0,Y 518.545,Z 400.74,A -85,B 0,C 180,E1 -4965.507,E2 -4965.507} C_VEL
LIN {X 0,Y 519.089,Z 388.106,A -85,B 0,C 180,E1 -4966.518,E2 -4966.518} C_VEL
LIN {X 0,Y 519.63,Z 374.449,A -85,B 0,C 180,E1 -4967.412,E2 -4967.412} C_VEL
LIN {X 0,Y 520.058,Z 361.268,A -85,B 0,C 180,E1 -4968.108,E2 -4968.108} C_VEL
LIN {X 0,Y 520.492,Z 346.122,A -85,B 0,C 180,E1 -4968.727,E2 -4968.727} C_VEL
LIN {X 0,Y 520.643,Z 331.135,A -85,B 0,C 180,E1 -4969.175,E2 -4969.175} C_VEL
LIN {X 0,Y 517.517,Z 319.905,A -85,B 0,C 180,E1 -4969.538,E2 -4969.538} C_VEL
LIN {X 0,Y 516.566,Z 316.56,A -85,B 0,C 180,E1 -4969.65,E2 -4969.65} C_VEL
LIN {X 0,Y 516.549,Z 312.485,A -85,B 0,C 180,E1 -4972.393,E2 -4972.393} C_VEL
LIN {X 0,Y 516.559,Z 308.725,A -85,B 0,C 180,E1 -4974.946,E2 -4974.946} C_VEL
LIN {X 0,Y 516.631,Z 304.595,A -85,B 0,C 180,E1 -4977.843,E2 -4977.843} C_VEL
LIN {X 0,Y 516.664,Z 301.395,A -85,B 0,C 180,E1 -4980.218,E2 -4980.218} C_VEL
LIN {X 0,Y 516.74,Z 297.692,A -85,B 0,C 180,E1 -4982.958,E2 -4982.958} C_VEL
LIN {X 0,Y 516.756,Z 293.776,A -85,B 0,C 180,E1 -4985.789,E2 -4985.789} C_VEL
LIN {X 0,Y 516.848,Z 289.45,A -85,B 0,C 180,E1 -4988.719,E2 -4988.719} C_VEL
LIN {X 0,Y 516.754,Z 286.821,A -85,B 0,C 180,E1 -4990.393,E2 -4990.393} C_VEL
LIN {X 0,Y 516.852,Z 286.728,A -85,B 0,C 180,E1 -4992.834,E2 -4992.834} C_VEL
LIN {X 0,Y 516.924,Z 286.723,A -85,B 0,C 180,E1 -4995.01,E2 -4995.01} C_VEL
LIN {X 0,Y 516.914,Z 286.724,A -85,B 0,C 180,E1 -4998.399,E2 -4998.399} C_VEL
LIN {X 0,Y 516.875,Z 286.723,A -85,B 0,C 180,E1 -5001.283,E2 -5001.283} C_VEL
LIN {X 0,Y 516.874,Z 286.725,A -85,B 0,C 180,E1 -5004.22,E2 -5004.22} C_VEL
LIN {X 0,Y 516.896,Z 286.725,A -85,B 0,C 180,E1 -5007.053,E2 -5007.053} C_VEL
LIN {X 0,Y 516.867,Z 286.724,A -85,B 0,C 180,E1 -5009.795,E2 -5009.795} C_VEL
LIN {X 0,Y 516.869,Z 286.725,A -85,B 0,C 180,E1 -5012.464,E2 -5012.464} C_VEL
LIN {X 0,Y 516.861,Z 286.727,A -85,B 0,C 180,E1 -5015.069,E2 -5015.069} C_VEL
LIN {X 0,Y 516.869,Z 286.722,A -85,B 0,C 180,E1 -5017.621,E2 -5017.621} C_VEL
LIN {X 0,Y 516.929,Z 286.72,A -85,B 0,C 180,E1 -5020.13,E2 -5020.13} C_VEL
LIN {X 0,Y 516.883,Z 286.721,A -85,B 0,C 180,E1 -5023.409,E2 -5023.409} C_VEL
LIN {X 0,Y 516.906,Z 286.721,A -85,B 0,C 180,E1 -5025.834,E2 -5025.834} C_VEL
LIN {X 0,Y 516.952,Z 286.713,A -85,B 0,C 180,E1 -5029.028,E2 -5029.028} C_VEL
LIN {X 0,Y 516.931,Z 286.718,A -85,B 0,C 180,E1 -5032.186,E2 -5032.186} C_VEL
LIN {X 0,Y 517.01,Z 286.702,A -85,B 0,C 180,E1 -5034.54,E2 -5034.54} C_VEL
LIN {X 0,Y 517.082,Z 286.697,A -85,B 0,C 180,E1 -5037.663,E2 -5037.663} C_VEL
LIN {X 0,Y 517.093,Z 286.696,A -85,B 0,C 180,E1 -5040.779,E2 -5040.779} C_VEL
LIN {X 0,Y 516.977,Z 286.712,A -85,B 0,C 180,E1 -5043.117,E2 -5043.117} C_VEL
LIN {X 0,Y 516.983,Z 286.706,A -85,B 0,C 180,E1 -5046.243,E2 -5046.243} C_VEL
LIN {X 0,Y 516.951,Z 286.713,A -85,B 0,C 180,E1 -5049.389,E2 -5049.389} C_VEL
LIN {X 0,Y 516.952,Z 286.712,A -85,B 0,C 180,E1 -5051.807,E2 -5051.807} C_VEL
LIN {X 0,Y 516.935,Z 286.72,A -85,B 0,C 180,E1 -5055.142,E2 -5055.142} C_VEL
LIN {X 0,Y 516.917,Z 286.719,A -85,B 0,C 180,E1 -5058.222,E2 -5058.222} C_VEL
LIN {X 0,Y 516.913,Z 286.717,A -85,B 0,C 180,E1 -5060.701,E2 -5060.701} C_VEL
LIN {X 0,Y 516.885,Z 286.724,A -85,B 0,C 180,E1 -5064.073,E2 -5064.073} C_VEL
LIN {X 0,Y 516.845,Z 286.727,A -85,B 0,C 180,E1 -5066.662,E2 -5066.662} C_VEL
LIN {X 0,Y 516.91,Z 286.72,A -85,B 0,C 180,E1 -5069.524,E2 -5069.524} C_VEL
LIN {X 0,Y 516.896,Z 286.721,A -85,B 0,C 180,E1 -5072.543,E2 -5072.543} C_VEL
LIN {X 0,Y 516.863,Z 286.73,A -85,B 0,C 180,E1 -5075.329,E2 -5075.329} C_VEL
LIN {X 0,Y 516.875,Z 286.725,A -85,B 0,C 180,E1 -5077.942,E2 -5077.942} C_VEL
LIN {X 0,Y 516.883,Z 286.724,A -85,B 0,C 180,E1 -5080.742,E2 -5080.742} C_VEL
LIN {X 0,Y 516.882,Z 286.722,A -85,B 0,C 180,E1 -5082.831,E2 -5082.831} C_VEL
LIN {X 0,Y 516.894,Z 286.722,A -85,B 0,C 180,E1 -5085.007,E2 -5085.007} C_VEL
LIN {X 0,Y 516.886,Z 286.725,A -85,B 0,C 180,E1 -5088.402,E2 -5088.402} C_VEL
LIN {X 0,Y 516.902,Z 286.797,A -85,B 0,C 180,E1 -5090.875,E2 -5090.875} C_VEL
LIN {X 0,Y 519.843,Z 298.25,A -85,B 0,C 180,E1 -5093.498,E2 -5093.498} C_VEL
LIN {X 0,Y 521.526,Z 305.227,A -85,B 0,C 180,E1 -5095.01,E2 -5095.01} C_VEL
LIN {X 0,Y 520.798,Z 317.626,A -85,B 0,C 180,E1 -5097.331,E2 -5097.331} C_VEL
LIN {X 0,Y 520.029,Z 332.408,A -85,B 0,C 180,E1 -5099.997,E2 -5099.997} C_VEL
LIN {X 0,Y 519.248,Z 349.838,A -85,B 0,C 180,E1 -5103.012,E2 -5103.012} C_VEL
LIN {X 0,Y 518.627,Z 367.758,A -85,B 0,C 180,E1 -5106.013,E2 -5106.013} C_VEL
LIN {X 0,Y 518.129,Z 384.736,A -85,B 0,C 180,E1 -5108.725,E2 -5108.725} C_VEL
LIN {X 0,Y 517.849,Z 395.594,A -85,B 0,C 180,E1 -5110.451,E2 -5110.451} C_VEL
LIN {X 0,Y 520.604,Z 411.006,A -85,B 0,C 180,E1 -5110.789,E2 -5110.789} C_VEL
LIN {X 0,Y 520.29,Z 426.877,A -85,B 0,C 180,E1 -5111.18,E2 -5111.18} C_VEL
LIN {X 0,Y 519.913,Z 441.989,A -85,B 0,C 180,E1 -5111.716,E2 -5111.716} C_VEL
LIN {X 0,Y 519.434,Z 456.267,A -85,B 0,C 180,E1 -5112.378,E2 -5112.378} C_VEL
LIN {X 0,Y 518.946,Z 469.909,A -85,B 0,C 180,E1 -5113.173,E2 -5113.173} C_VEL
LIN {X 0,Y 518.532,Z 483.019,A -85,B 0,C 180,E1 -5114.109,E2 -5114.109} C_VEL
LIN {X 0,Y 518.017,Z 495.351,A -85,B 0,C 180,E1 -5115.163,E2 -5115.163} C_VEL
LIN {X 0,Y 517.609,Z 506.117,A -85,B 0,C 180,E1 -5116.255,E2 -5116.255} C_VEL
LIN {X 0,Y 517.26,Z 516.106,A -85,B 0,C 180,E1 -5117.444,E2 -5117.444} C_VEL
LIN {X 0,Y 516.994,Z 524.581,A -85,B 0,C 180,E1 -5118.632,E2 -5118.632} C_VEL
LIN {X 0,Y 516.71,Z 532.73,A -85,B 0,C 180,E1 -5120.014,E2 -5120.014} C_VEL
LIN {X 0,Y 516.541,Z 539.421,A -85,B 0,C 180,E1 -5121.393,E2 -5121.393} C_VEL
LIN {X 0,Y 516.391,Z 545.604,A -85,B 0,C 180,E1 -5122.964,E2 -5122.964} C_VEL
LIN {X 0,Y 516.374,Z 550.385,A -85,B 0,C 180,E1 -5124.533,E2 -5124.533} C_VEL
LIN {X 0,Y 516.307,Z 553.887,A -85,B 0,C 180,E1 -5126.098,E2 -5126.098} C_VEL
LIN {X 0,Y 516.258,Z 556.19,A -85,B 0,C 180,E1 -5127.66,E2 -5127.66} C_VEL
LIN {X 0,Y 516.158,Z 557.348,A -85,B 0,C 180,E1 -5129.22,E2 -5129.22} C_VEL
LIN {X 0,Y 516.158,Z 557.346,A -85,B 0,C 180,E1 -5130.78,E2 -5130.78} C_VEL
LIN {X 0,Y 516.258,Z 556.185,A -85,B 0,C 180,E1 -5132.341,E2 -5132.341} C_VEL
LIN {X 0,Y 516.307,Z 553.882,A -85,B 0,C 180,E1 -5133.903,E2 -5133.903} C_VEL
LIN {X 0,Y 516.374,Z 550.386,A -85,B 0,C 180,E1 -5135.467,E2 -5135.467} C_VEL
LIN {X 0,Y 516.396,Z 545.609,A -85,B 0,C 180,E1 -5137.036,E2 -5137.036} C_VEL
LIN {X 0,Y 516.541,Z 539.418,A -85,B 0,C 180,E1 -5138.608,E2 -5138.608} C_VEL
LIN {X 0,Y 516.757,Z 531.64,A -85,B 0,C 180,E1 -5140.184,E2 -5140.184} C_VEL
LIN {X 0,Y 517,Z 523.292,A -85,B 0,C 180,E1 -5141.567,E2 -5141.567} C_VEL
LIN {X 0,Y 517.308,Z 514.55,A -85,B 0,C 180,E1 -5142.754,E2 -5142.754} C_VEL
LIN {X 0,Y 517.688,Z 504.174,A -85,B 0,C 180,E1 -5143.944,E2 -5143.944} C_VEL
LIN {X 0,Y 518.125,Z 491.976,A -85,B 0,C 180,E1 -5145.123,E2 -5145.123} C_VEL
LIN {X 0,Y 518.61,Z 479.505,A -85,B 0,C 180,E1 -5146.13,E2 -5146.13} C_VEL
LIN {X 0,Y 519.038,Z 466.133,A -85,B 0,C 180,E1 -5147.027,E2 -5147.027} C_VEL
LIN {X 0,Y 519.501,Z 451.482,A -85,B 0,C 180,E1 -5147.823,E2 -5147.823} C_VEL
LIN {X 0,Y 519.962,Z 436.736,A -85,B 0,C 180,E1 -5148.451,E2 -5148.451} C_VEL
LIN {X 0,Y 520.289,Z 421.299,A -85,B 0,C 180,E1 -5148.941,E2 -5148.941} C_VEL
LIN {X 0,Y 520.408,Z 409.786,A -85,B 0,C 180,E1 -5149.207,E2 -5149.207} C_VEL
LIN {X 0,Y 517.944,Z 396.574,A -85,B 0,C 180,E1 -5149.489,E2 -5149.489} C_VEL
LIN {X 0,Y 517.771,Z 394.731,A -85,B 0,C 180,E1 -5149.553,E2 -5149.553} C_VEL
LIN {X 0,Y 518.144,Z 378.132,A -85,B 0,C 180,E1 -5152.111,E2 -5152.111} C_VEL
LIN {X 0,Y 518.484,Z 361.993,A -85,B 0,C 180,E1 -5154.65,E2 -5154.65} C_VEL
LIN {X 0,Y 519.001,Z 345.377,A -85,B 0,C 180,E1 -5157.414,E2 -5157.414} C_VEL
LIN {X 0,Y 519.728,Z 330.502,A -85,B 0,C 180,E1 -5160.067,E2 -5160.067} C_VEL
LIN {X 0,Y 520.713,Z 317.224,A -85,B 0,C 180,E1 -5162.675,E2 -5162.675} C_VEL
LIN {X 0,Y 521.839,Z 307.71,A -85,B 0,C 180,E1 -5164.762,E2 -5164.762} C_VEL
LIN {X 0,Y 521.321,Z 303.749,A -85,B 0,C 180,E1 -5165.832,E2 -5165.832} C_VEL
LIN {X 0,Y 519.653,Z 297.539,A -85,B 0,C 180,E1 -5167.88,E2 -5167.88} C_VEL
LIN {X 0,Y 518.621,Z 293.442,A -85,B 0,C 180,E1 -5169.562,E2 -5169.562} C_VEL
LIN {X 0,Y 517.621,Z 289.636,A -85,B 0,C 180,E1 -5171.706,E2 -5171.706} C_VEL
LIN {X 0,Y 517.276,Z 288.289,A -85,B 0,C 180,E1 -5172.805,E2 -5172.805} C_VEL
LIN {X 0,Y 516.905,Z 286.726,A -85,B 0,C 180,E1 -5175.116,E2 -5175.116} C_VEL
LIN {X 0,Y 516.915,Z 286.789,A -85,B 0,C 180,E1 -5178.399,E2 -5178.399} C_VEL
LIN {X 0,Y 517.168,Z 288.359,A -85,B 0,C 180,E1 -5181.31,E2 -5181.31} C_VEL
LIN {X 0,Y 517.371,Z 289.839,A -85,B 0,C 180,E1 -5183.295,E2 -5183.295} C_VEL
LIN {X 0,Y 517.435,Z 292.221,A -85,B 0,C 180,E1 -5186.16,E2 -5186.16} C_VEL
LIN {X 0,Y 517.24,Z 294.605,A -85,B 0,C 180,E1 -5188.914,E2 -5188.914} C_VEL
LIN {X 0,Y 517.196,Z 296.854,A -85,B 0,C 180,E1 -5191.601,E2 -5191.601} C_VEL
LIN {X 0,Y 517.099,Z 299.064,A -85,B 0,C 180,E1 -5194.22,E2 -5194.22} C_VEL
LIN {X 0,Y 517.007,Z 301.176,A -85,B 0,C 180,E1 -5196.783,E2 -5196.783} C_VEL
LIN {X 0,Y 516.913,Z 303.664,A -85,B 0,C 180,E1 -5199.741,E2 -5199.741} C_VEL
LIN {X 0,Y 516.785,Z 306.111,A -85,B 0,C 180,E1 -5202.591,E2 -5202.591} C_VEL
LIN {X 0,Y 516.777,Z 308.246,A -85,B 0,C 180,E1 -5205.025,E2 -5205.025} C_VEL
LIN {X 0,Y 516.691,Z 309.198,A -85,B 0,C 180,E1 -5206.054,E2 -5206.054} C_VEL
LIN {X 0,Y 518.825,Z 316.317,A -85,B 0,C 180,E1 -5206.325,E2 -5206.325} C_VEL
LIN {X 0,Y 518.876,Z 325.339,A -85,B 0,C 180,E1 -5206.638,E2 -5206.638} C_VEL
LIN {X 0,Y 518.596,Z 337.905,A -85,B 0,C 180,E1 -5207.209,E2 -5207.209} C_VEL
LIN {X 0,Y 518.344,Z 349.835,A -85,B 0,C 180,E1 -5207.922,E2 -5207.922} C_VEL
LIN {X 0,Y 518.016,Z 359.65,A -85,B 0,C 180,E1 -5208.655,E2 -5208.655} C_VEL
LIN {X 0,Y 517.644,Z 370.228,A -85,B 0,C 180,E1 -5209.636,E2 -5209.636} C_VEL
LIN {X 0,Y 517.428,Z 378.825,A -85,B 0,C 180,E1 -5210.62,E2 -5210.62} C_VEL
LIN {X 0,Y 517.132,Z 387.243,A -85,B 0,C 180,E1 -5211.796,E2 -5211.796} C_VEL
LIN {X 0,Y 516.931,Z 393.949,A -85,B 0,C 180,E1 -5212.972,E2 -5212.972} C_VEL
LIN {X 0,Y 516.767,Z 399.312,A -85,B 0,C 180,E1 -5214.146,E2 -5214.146} C_VEL
LIN {X 0,Y 516.597,Z 403.521,A -85,B 0,C 180,E1 -5215.318,E2 -5215.318} C_VEL
LIN {X 0,Y 516.588,Z 405.72,A -85,B 0,C 180,E1 -5216.1,E2 -5216.1} C_VEL
LIN {X 0,Y 516.624,Z 407.499,A -85,B 0,C 180,E1 -5216.881,E2 -5216.881} C_VEL
LIN {X 0,Y 516.498,Z 408.868,A -85,B 0,C 180,E1 -5217.661,E2 -5217.661} C_VEL
LIN {X 0,Y 516.446,Z 410.381,A -85,B 0,C 180,E1 -5219.22,E2 -5219.22} C_VEL
LIN {X 0,Y 516.436,Z 410.57,A -85,B 0,C 180,E1 -5220,E2 -5220} C_VEL
LIN {X 0,Y 516.424,Z 410.359,A -85,B 0,C 180,E1 -5220.78,E2 -5220.78} C_VEL
LIN {X 0,Y 516.416,Z 408.761,A -85,B 0,C 180,E1 -5222.34,E2 -5222.34} C_VEL
LIN {X 0,Y 516.483,Z 407.371,A -85,B 0,C 180,E1 -5223.12,E2 -5223.12} C_VEL
LIN {X 0,Y 516.579,Z 404.474,A -85,B 0,C 180,E1 -5224.291,E2 -5224.291} C_VEL
LIN {X 0,Y 516.571,Z 400.585,A -85,B 0,C 180,E1 -5225.465,E2 -5225.465} C_VEL
LIN {X 0,Y 516.729,Z 395.336,A -85,B 0,C 180,E1 -5226.681,E2 -5226.681} C_VEL
LIN {X 0,Y 516.882,Z 389.247,A -85,B 0,C 180,E1 -5227.815,E2 -5227.815} C_VEL
LIN {X 0,Y 517.114,Z 381.359,A -85,B 0,C 180,E1 -5228.992,E2 -5228.992} C_VEL
LIN {X 0,Y 517.311,Z 373.318,A -85,B 0,C 180,E1 -5229.975,E2 -5229.975} C_VEL
LIN {X 0,Y 517.672,Z 363.5,A -85,B 0,C 180,E1 -5230.957,E2 -5230.957} C_VEL
LIN {X 0,Y 517.896,Z 353.901,A -85,B 0,C 180,E1 -5231.745,E2 -5231.745} C_VEL
LIN {X 0,Y 518.196,Z 341.867,A -85,B 0,C 180,E1 -5232.533,E2 -5232.533} C_VEL
LIN {X 0,Y 518.499,Z 329.096,A -85,B 0,C 180,E1 -5233.173,E2 -5233.173} C_VEL
LIN {X 0,Y 518.513,Z 316.265,A -85,B 0,C 180,E1 -5233.646,E2 -5233.646} C_VEL
LIN {X 0,Y 516.41,Z 306.806,A -85,B 0,C 180,E1 -5233.979,E2 -5233.979} C_VEL
LIN {X 0,Y 516.372,Z 303.985,A -85,B 0,C 180,E1 -5236.608,E2 -5236.608} C_VEL
LIN {X 0,Y 516.444,Z 300.465,A -85,B 0,C 180,E1 -5239.89,E2 -5239.89} C_VEL
LIN {X 0,Y 516.454,Z 296.893,A -85,B 0,C 180,E1 -5243.243,E2 -5243.243} C_VEL
LIN {X 0,Y 516.489,Z 293.844,A -85,B 0,C 180,E1 -5246.093,E2 -5246.093} C_VEL
LIN {X 0,Y 516.533,Z 291.314,A -85,B 0,C 180,E1 -5248.439,E2 -5248.439} C_VEL
LIN {X 0,Y 516.516,Z 288.409,A -85,B 0,C 180,E1 -5251.135,E2 -5251.135} C_VEL
LIN {X 0,Y 516.485,Z 287.006,A -85,B 0,C 180,E1 -5252.471,E2 -5252.471} C_VEL
LIN {X 0,Y 516.787,Z 286.74,A -85,B 0,C 180,E1 -5254.832,E2 -5254.832} C_VEL
LIN {X 0,Y 516.884,Z 286.722,A -85,B 0,C 180,E1 -5257.943,E2 -5257.943} C_VEL
LIN {X 0,Y 516.886,Z 286.727,A -85,B 0,C 180,E1 -5260.742,E2 -5260.742} C_VEL
LIN {X 0,Y 516.876,Z 286.724,A -85,B 0,C 180,E1 -5262.948,E2 -5262.948} C_VEL
LIN {X 0,Y 516.883,Z 286.727,A -85,B 0,C 180,E1 -5266.107,E2 -5266.107} C_VEL
LIN {X 0,Y 516.86,Z 286.728,A -85,B 0,C 180,E1 -5266.344,E2 -5266.344} C_VEL
LIN {X 0,Y 516.152,Z 286.855,A -85,B 0,C 180,E1 -5266.996,E2 -5266.996} C_VEL
LIN {X 0,Y 513.241,Z 287.183,A -85,B 0,C 180,E1 -5268.056,E2 -5268.056} C_VEL
LIN {X 0,Y 510.816,Z 287.481,A -85,B 0,C 180,E1 -5268.906,E2 -5268.906} C_VEL
LIN {X 0,Y 509.732,Z 287.753,A -85,B 0,C 180,E1 -5269.669,E2 -5269.669} C_VEL
LIN {X 0,Y 509.714,Z 287.89,A -85,B 0,C 180,E1 -5269.778,E2 -5269.778} C_VEL
LIN {X 0,Y 509.788,Z 290.963,A -85,B 0,C 180,E1 -5271.796,E2 -5271.796} C_VEL
LIN {X 0,Y 509.714,Z 295.08,A -85,B 0,C 180,E1 -5274.612,E2 -5274.612} C_VEL
LIN {X 0,Y 509.716,Z 298.988,A -85,B 0,C 180,E1 -5277.47,E2 -5277.47} C_VEL
LIN {X 0,Y 509.599,Z 302.843,A -85,B 0,C 180,E1 -5280.325,E2 -5280.325} C_VEL
LIN {X 0,Y 509.545,Z 306.368,A -85,B 0,C 180,E1 -5282.925,E2 -5282.925} C_VEL
LIN {X 0,Y 509.519,Z 310.1,A -85,B 0,C 180,E1 -5285.556,E2 -5285.556} C_VEL
LIN {X 0,Y 509.473,Z 313.975,A -85,B 0,C 180,E1 -5288.133,E2 -5288.133} C_VEL
LIN {X 0,Y 509.511,Z 317.028,A -85,B 0,C 180,E1 -5290.172,E2 -5290.172} C_VEL
LIN {X 0,Y 513.512,Z 330.566,A -85,B 0,C 180,E1 -5290.611,E2 -5290.611} C_VEL
LIN {X 0,Y 514.087,Z 334.253,A -85,B 0,C 180,E1 -5290.726,E2 -5290.726} C_VEL
LIN {X 0,Y 513.791,Z 349.061,A -85,B 0,C 180,E1 -5291.196,E2 -5291.196} C_VEL
LIN {X 0,Y 513.259,Z 364.243,A -85,B 0,C 180,E1 -5291.849,E2 -5291.849} C_VEL
LIN {X 0,Y 512.735,Z 378.596,A -85,B 0,C 180,E1 -5292.655,E2 -5292.655} C_VEL
LIN {X 0,Y 512.194,Z 391.583,A -85,B 0,C 180,E1 -5293.561,E2 -5293.561} C_VEL
LIN {X 0,Y 511.616,Z 403.74,A -85,B 0,C 180,E1 -5294.587,E2 -5294.587} C_VEL
LIN {X 0,Y 511.012,Z 416.291,A -85,B 0,C 180,E1 -5295.87,E2 -5295.87} C_VEL
LIN {X 0,Y 510.538,Z 426.133,A -85,B 0,C 180,E1 -5297.074,E2 -5297.074} C_VEL
LIN {X 0,Y 510.112,Z 435.944,A -85,B 0,C 180,E1 -5298.512,E2 -5298.512} C_VEL
LIN {X 0,Y 509.803,Z 443.68,A -85,B 0,C 180,E1 -5299.876,E2 -5299.876} C_VEL
LIN {X 0,Y 509.558,Z 450.256,A -85,B 0,C 180,E1 -5301.273,E2 -5301.273} C_VEL
LIN {X 0,Y 509.395,Z 456.338,A -85,B 0,C 180,E1 -5302.867,E2 -5302.867} C_VEL
LIN {X 0,Y 509.316,Z 461.039,A -85,B 0,C 180,E1 -5304.457,E2 -5304.457} C_VEL
LIN {X 0,Y 509.236,Z 464.49,A -85,B 0,C 180,E1 -5306.043,E2 -5306.043} C_VEL
LIN {X 0,Y 509.189,Z 466.769,A -85,B 0,C 180,E1 -5307.627,E2 -5307.627} C_VEL
LIN {X 0,Y 509.089,Z 467.936,A -85,B 0,C 180,E1 -5309.209,E2 -5309.209} C_VEL
LIN {X 0,Y 509.09,Z 467.954,A -85,B 0,C 180,E1 -5310.791,E2 -5310.791} C_VEL
LIN {X 0,Y 509.19,Z 466.853,A -85,B 0,C 180,E1 -5312.373,E2 -5312.373} C_VEL
LIN {X 0,Y 509.236,Z 464.645,A -85,B 0,C 180,E1 -5313.957,E2 -5313.957} C_VEL
LIN {X 0,Y 509.314,Z 461.273,A -85,B 0,C 180,E1 -5315.543,E2 -5315.543} C_VEL
LIN {X 0,Y 509.394,Z 456.652,A -85,B 0,C 180,E1 -5317.133,E2 -5317.133} C_VEL
LIN {X 0,Y 509.54,Z 450.648,A -85,B 0,C 180,E1 -5318.727,E2 -5318.727} C_VEL
LIN {X 0,Y 509.807,Z 443.084,A -85,B 0,C 180,E1 -5320.324,E2 -5320.324} C_VEL
LIN {X 0,Y 510.14,Z 435.511,A -85,B 0,C 180,E1 -5321.647,E2 -5321.647} C_VEL
LIN {X 0,Y 510.499,Z 426.785,A -85,B 0,C 180,E1 -5322.927,E2 -5322.927} C_VEL
LIN {X 0,Y 510.998,Z 417.057,A -85,B 0,C 180,E1 -5324.13,E2 -5324.13} C_VEL
LIN {X 0,Y 511.503,Z 405.745,A -85,B 0,C 180,E1 -5325.312,E2 -5325.312} C_VEL
LIN {X 0,Y 512.063,Z 394.441,A -85,B 0,C 180,E1 -5326.3,E2 -5326.3} C_VEL
LIN {X 0,Y 512.621,Z 381.454,A -85,B 0,C 180,E1 -5327.246,E2 -5327.246} C_VEL
LIN {X 0,Y 513.097,Z 367.843,A -85,B 0,C 180,E1 -5328.053,E2 -5328.053} C_VEL
LIN {X 0,Y 513.651,Z 354.073,A -85,B 0,C 180,E1 -5328.695,E2 -5328.695} C_VEL
LIN {X 0,Y 514,Z 339.497,A -85,B 0,C 180,E1 -5329.213,E2 -5329.213} C_VEL
LIN {X 0,Y 513.941,Z 332.438,A -85,B 0,C 180,E1 -5329.416,E2 -5329.416} C_VEL
LIN {X 0,Y 510.953,Z 321.693,A -85,B 0,C 180,E1 -5329.774,E2 -5329.774} C_VEL
LIN {X 0,Y 509.549,Z 316.984,A -85,B 0,C 180,E1 -5329.932,E2 -5329.932} C_VEL
LIN {X 0,Y 509.487,Z 312.808,A -85,B 0,C 180,E1 -5332.721,E2 -5332.721} C_VEL
LIN {X 0,Y 509.507,Z 308.987,A -85,B 0,C 180,E1 -5335.316,E2 -5335.316} C_VEL
LIN {X 0,Y 509.592,Z 305.173,A -85,B 0,C 180,E1 -5338.036,E2 -5338.036} C_VEL
LIN {X 0,Y 509.64,Z 300.864,A -85,B 0,C 180,E1 -5341.241,E2 -5341.241} C_VEL
LIN {X 0,Y 509.702,Z 297.857,A -85,B 0,C 180,E1 -5343.472,E2 -5343.472} C_VEL
LIN {X 0,Y 509.728,Z 293.833,A -85,B 0,C 180,E1 -5346.361,E2 -5346.361} C_VEL
LIN {X 0,Y 509.799,Z 289.373,A -85,B 0,C 180,E1 -5349.357,E2 -5349.357} C_VEL
LIN {X 0,Y 509.716,Z 287.758,A -85,B 0,C 180,E1 -5350.394,E2 -5350.394} C_VEL
LIN {X 0,Y 509.799,Z 287.608,A -85,B 0,C 180,E1 -5353.059,E2 -5353.059} C_VEL
LIN {X 0,Y 509.831,Z 287.604,A -85,B 0,C 180,E1 -5355.792,E2 -5355.792} C_VEL
LIN {X 0,Y 509.856,Z 287.602,A -85,B 0,C 180,E1 -5358.574,E2 -5358.574} C_VEL
LIN {X 0,Y 509.848,Z 287.602,A -85,B 0,C 180,E1 -5361.787,E2 -5361.787} C_VEL
LIN {X 0,Y 509.834,Z 287.602,A -85,B 0,C 180,E1 -5364.622,E2 -5364.622} C_VEL
LIN {X 0,Y 509.862,Z 287.599,A -85,B 0,C 180,E1 -5367.481,E2 -5367.481} C_VEL
LIN {X 0,Y 509.853,Z 287.6,A -85,B 0,C 180,E1 -5370.275,E2 -5370.275} C_VEL
LIN {X 0,Y 509.822,Z 287.602,A -85,B 0,C 180,E1 -5372.941,E2 -5372.941} C_VEL
LIN {X 0,Y 509.846,Z 287.603,A -85,B 0,C 180,E1 -5375.573,E2 -5375.573} C_VEL
LIN {X 0,Y 509.822,Z 287.6,A -85,B 0,C 180,E1 -5378.149,E2 -5378.149} C_VEL
LIN {X 0,Y 509.855,Z 287.6,A -85,B 0,C 180,E1 -5380.681,E2 -5380.681} C_VEL
LIN {X 0,Y 509.852,Z 287.595,A -85,B 0,C 180,E1 -5383.174,E2 -5383.174} C_VEL
LIN {X 0,Y 509.874,Z 287.598,A -85,B 0,C 180,E1 -5385.634,E2 -5385.634} C_VEL
LIN {X 0,Y 509.914,Z 287.591,A -85,B 0,C 180,E1 -5388.874,E2 -5388.874} C_VEL
LIN {X 0,Y 509.884,Z 287.597,A -85,B 0,C 180,E1 -5392.077,E2 -5392.077} C_VEL
LIN {X 0,Y 509.961,Z 287.579,A -85,B 0,C 180,E1 -5394.464,E2 -5394.464} C_VEL
LIN {X 0,Y 510.053,Z 287.573,A -85,B 0,C 180,E1 -5397.631,E2 -5397.631} C_VEL
LIN {X 0,Y 510.058,Z 287.569,A -85,B 0,C 180,E1 -5400,E2 -5400} C_VEL
LIN {X 0,Y 510.049,Z 287.576,A -85,B 0,C 180,E1 -5402.369,E2 -5402.369} C_VEL
LIN {X 0,Y 509.937,Z 287.584,A -85,B 0,C 180,E1 -5406.33,E2 -5406.33} C_VEL
LIN {X 0,Y 509.908,Z 287.595,A -85,B 0,C 180,E1 -5408.72,E2 -5408.72} C_VEL
LIN {X 0,Y 509.905,Z 287.592,A -85,B 0,C 180,E1 -5411.932,E2 -5411.932} C_VEL
LIN {X 0,Y 509.895,Z 287.594,A -85,B 0,C 180,E1 -5415.242,E2 -5415.242} C_VEL
LIN {X 0,Y 509.862,Z 287.601,A -85,B 0,C 180,E1 -5418.484,E2 -5418.484} C_VEL
LIN {X 0,Y 509.851,Z 287.595,A -85,B 0,C 180,E1 -5421.002,E2 -5421.002} C_VEL
LIN {X 0,Y 509.819,Z 287.607,A -85,B 0,C 180,E1 -5423.564,E2 -5423.564} C_VEL
LIN {X 0,Y 509.834,Z 287.598,A -85,B 0,C 180,E1 -5426.361,E2 -5426.361} C_VEL
LIN {X 0,Y 509.85,Z 287.602,A -85,B 0,C 180,E1 -5428.846,E2 -5428.846} C_VEL
LIN {X 0,Y 509.82,Z 287.605,A -85,B 0,C 180,E1 -5431.59,E2 -5431.59} C_VEL
LIN {X 0,Y 509.846,Z 287.599,A -85,B 0,C 180,E1 -5434.414,E2 -5434.414} C_VEL
LIN {X 0,Y 509.805,Z 287.607,A -85,B 0,C 180,E1 -5437.342,E2 -5437.342} C_VEL
LIN {X 0,Y 509.837,Z 287.605,A -85,B 0,C 180,E1 -5440.382,E2 -5440.382} C_VEL
LIN {X 0,Y 509.822,Z 287.602,A -85,B 0,C 180,E1 -5443.062,E2 -5443.062} C_VEL
LIN {X 0,Y 509.821,Z 287.601,A -85,B 0,C 180,E1 -5445.793,E2 -5445.793} C_VEL
LIN {X 0,Y 509.832,Z 287.605,A -85,B 0,C 180,E1 -5448.572,E2 -5448.572} C_VEL
LIN {X 0,Y 509.848,Z 287.73,A -85,B 0,C 180,E1 -5450.446,E2 -5450.446} C_VEL
LIN {X 0,Y 513.161,Z 300.582,A -85,B 0,C 180,E1 -5453.434,E2 -5453.434} C_VEL
LIN {X 0,Y 514.797,Z 307.787,A -85,B 0,C 180,E1 -5455.014,E2 -5455.014} C_VEL
LIN {X 0,Y 513.911,Z 321.117,A -85,B 0,C 180,E1 -5457.537,E2 -5457.537} C_VEL
LIN {X 0,Y 512.995,Z 338.505,A -85,B 0,C 180,E1 -5460.697,E2 -5460.697} C_VEL
LIN {X 0,Y 512.091,Z 357.161,A -85,B 0,C 180,E1 -5463.949,E2 -5463.949} C_VEL
LIN {X 0,Y 511.403,Z 375.494,A -85,B 0,C 180,E1 -5467.036,E2 -5467.036} C_VEL
LIN {X 0,Y 510.851,Z 394.304,A -85,B 0,C 180,E1 -5470.093,E2 -5470.093} C_VEL
LIN {X 0,Y 510.839,Z 395.162,A -85,B 0,C 180,E1 -5470.217,E2 -5470.217} C_VEL
LIN {X 0,Y 513.441,Z 409.677,A -85,B 0,C 180,E1 -5470.537,E2 -5470.537} C_VEL
LIN {X 0,Y 513.7,Z 414.03,A -85,B 0,C 180,E1 -5470.64,E2 -5470.64} C_VEL
LIN {X 0,Y 513.335,Z 429.706,A -85,B 0,C 180,E1 -5471.071,E2 -5471.071} C_VEL
LIN {X 0,Y 512.881,Z 445.426,A -85,B 0,C 180,E1 -5471.681,E2 -5471.681} C_VEL
LIN {X 0,Y 512.361,Z 460.285,A -85,B 0,C 180,E1 -5472.436,E2 -5472.436} C_VEL
LIN {X 0,Y 511.888,Z 473.042,A -85,B 0,C 180,E1 -5473.243,E2 -5473.243} C_VEL
LIN {X 0,Y 511.371,Z 486.577,A -85,B 0,C 180,E1 -5474.28,E2 -5474.28} C_VEL
LIN {X 0,Y 510.874,Z 498.306,A -85,B 0,C 180,E1 -5475.358,E2 -5475.358} C_VEL
LIN {X 0,Y 510.408,Z 510.22,A -85,B 0,C 180,E1 -5476.666,E2 -5476.666} C_VEL
LIN {X 0,Y 509.968,Z 520.867,A -85,B 0,C 180,E1 -5478.07,E2 -5478.07} C_VEL
LIN {X 0,Y 509.786,Z 529.746,A -85,B 0,C 180,E1 -5479.475,E2 -5479.475} C_VEL
LIN {X 0,Y 509.516,Z 537.114,A -85,B 0,C 180,E1 -5480.873,E2 -5480.873} C_VEL
LIN {X 0,Y 509.351,Z 543.957,A -85,B 0,C 180,E1 -5482.468,E2 -5482.468} C_VEL
LIN {X 0,Y 509.275,Z 549.264,A -85,B 0,C 180,E1 -5484.059,E2 -5484.059} C_VEL
LIN {X 0,Y 509.158,Z 552.277,A -85,B 0,C 180,E1 -5485.25,E2 -5485.25} C_VEL
LIN {X 0,Y 509.188,Z 555.183,A -85,B 0,C 180,E1 -5486.835,E2 -5486.835} C_VEL
LIN {X 0,Y 509.11,Z 556.909,A -85,B 0,C 180,E1 -5488.418,E2 -5488.418} C_VEL
LIN {X 0,Y 509.062,Z 557.5,A -85,B 0,C 180,E1 -5490,E2 -5490} C_VEL
LIN {X 0,Y 509.11,Z 556.906,A -85,B 0,C 180,E1 -5491.582,E2 -5491.582} C_VEL
LIN {X 0,Y 509.188,Z 555.177,A -85,B 0,C 180,E1 -5493.165,E2 -5493.165} C_VEL
LIN {X 0,Y 509.159,Z 552.274,A -85,B 0,C 180,E1 -5494.751,E2 -5494.751} C_VEL
LIN {X 0,Y 509.306,Z 548.079,A -85,B 0,C 180,E1 -5496.338,E2 -5496.338} C_VEL
LIN {X 0,Y 509.385,Z 542.399,A -85,B 0,C 180,E1 -5497.931,E2 -5497.931} C_VEL
LIN {X 0,Y 509.536,Z 535.095,A -85,B 0,C 180,E1 -5499.527,E2 -5499.527} C_VEL
LIN {X 0,Y 509.857,Z 527.296,A -85,B 0,C 180,E1 -5500.926,E2 -5500.926} C_VEL
LIN {X 0,Y 510.125,Z 517.859,A -85,B 0,C 180,E1 -5502.33,E2 -5502.33} C_VEL
LIN {X 0,Y 510.543,Z 506.484,A -85,B 0,C 180,E1 -5503.737,E2 -5503.737} C_VEL
LIN {X 0,Y 510.974,Z 494.772,A -85,B 0,C 180,E1 -5504.945,E2 -5504.945} C_VEL
LIN {X 0,Y 511.492,Z 481.904,A -85,B 0,C 180,E1 -5506.053,E2 -5506.053} C_VEL
LIN {X 0,Y 511.961,Z 469.246,A -85,B 0,C 180,E1 -5506.961,E2 -5506.961} C_VEL
LIN {X 0,Y 512.432,Z 455.564,A -85,B 0,C 180,E1 -5507.768,E2 -5507.768} C_VEL
LIN {X 0,Y 512.963,Z 441.206,A -85,B 0,C 180,E1 -5508.445,E2 -5508.445} C_VEL
LIN {X 0,Y 513.324,Z 425.731,A -85,B 0,C 180,E1 -5509.004,E2 -5509.004} C_VEL
LIN {X 0,Y 513.558,Z 410.947,A -85,B 0,C 180,E1 -5509.382,E2 -5509.382} C_VEL
LIN {X 0,Y 511.157,Z 397.66,A -85,B 0,C 180,E1 -5509.686,E2 -5509.686} C_VEL
LIN {X 0,Y 510.748,Z 394.088,A -85,B 0,C 180,E1 -5509.754,E2 -5509.754} C_VEL
LIN {X 0,Y 511.171,Z 375.673,A -85,B 0,C 180,E1 -5512.642,E2 -5512.642} C_VEL
LIN {X 0,Y 511.594,Z 358.658,A -85,B 0,C 180,E1 -5515.423,E2 -5515.423} C_VEL
LIN {X 0,Y 512.216,Z 343.567,A -85,B 0,C 180,E1 -5518.03,E2 -5518.03} C_VEL
LIN {X 0,Y 512.934,Z 330.453,A -85,B 0,C 180,E1 -5520.462,E2 -5520.462} C_VEL
LIN {X 0,Y 514.012,Z 318.374,A -85,B 0,C 180,E1 -5522.922,E2 -5522.922} C_VEL
LIN {X 0,Y 515.139,Z 309.399,A -85,B 0,C 180,E1 -5524.96,E2 -5524.96} C_VEL
LIN {X 0,Y 514.566,Z 305.8,A -85,B 0,C 180,E1 -5525.966,E2 -5525.966} C_VEL
LIN {X 0,Y 512.921,Z 299.618,A -85,B 0,C 180,E1 -5528.068,E2 -5528.068} C_VEL
LIN {X 0,Y 511.902,Z 295.671,A -85,B 0,C 180,E1 -5529.751,E2 -5529.751} C_VEL
LIN {X 0,Y 511.156,Z 292.845,A -85,B 0,C 180,E1 -5531.297,E2 -5531.297} C_VEL
LIN {X 0,Y 510.417,Z 290.147,A -85,B 0,C 180,E1 -5533.508,E2 -5533.508} C_VEL
LIN {X 0,Y 510.146,Z 288.848,A -85,B 0,C 180,E1 -5535.756,E2 -5535.756} C_VEL
LIN {X 0,Y 510.139,Z 288.93,A -85,B 0,C 180,E1 -5538.603,E2 -5538.603} C_VEL
LIN {X 0,Y 510.263,Z 289.809,A -85,B 0,C 180,E1 -5540.686,E2 -5540.686} C_VEL
LIN {X 0,Y 510.443,Z 291.277,A -85,B 0,C 180,E1 -5542.994,E2 -5542.994} C_VEL
LIN {X 0,Y 510.476,Z 293.345,A -85,B 0,C 180,E1 -5545.696,E2 -5545.696} C_VEL
LIN {X 0,Y 510.305,Z 295.762,A -85,B 0,C 180,E1 -5548.636,E2 -5548.636} C_VEL
LIN {X 0,Y 510.212,Z 298.374,A -85,B 0,C 180,E1 -5551.834,E2 -5551.834} C_VEL
LIN {X 0,Y 510.085,Z 300.745,A -85,B 0,C 180,E1 -5554.715,E2 -5554.715} C_VEL
LIN {X 0,Y 510.001,Z 302.952,A -85,B 0,C 180,E1 -5557.412,E2 -5557.412} C_VEL
LIN {X 0,Y 509.865,Z 305.689,A -85,B 0,C 180,E1 -5560.682,E2 -5560.682} C_VEL
LIN {X 0,Y 509.765,Z 307.824,A -85,B 0,C 180,E1 -5563.171,E2 -5563.171} C_VEL
LIN {X 0,Y 509.696,Z 310.193,A -85,B 0,C 180,E1 -5565.82,E2 -5565.82} C_VEL
LIN {X 0,Y 512.201,Z 318.25,A -85,B 0,C 180,E1 -5566.144,E2 -5566.144} C_VEL
LIN {X 0,Y 512.012,Z 330.785,A -85,B 0,C 180,E1 -5566.617,E2 -5566.617} C_VEL
LIN {X 0,Y 511.73,Z 342.089,A -85,B 0,C 180,E1 -5567.188,E2 -5567.188} C_VEL
LIN {X 0,Y 511.41,Z 353.912,A -85,B 0,C 180,E1 -5567.959,E2 -5567.959} C_VEL
LIN {X 0,Y 511.071,Z 364.246,A -85,B 0,C 180,E1 -5568.8,E2 -5568.8} C_VEL
LIN {X 0,Y 510.74,Z 373.26,A -85,B 0,C 180,E1 -5569.695,E2 -5569.695} C_VEL
LIN {X 0,Y 510.436,Z 381.524,A -85,B 0,C 180,E1 -5570.69,E2 -5570.69} C_VEL
LIN {X 0,Y 510.095,Z 389.567,A -85,B 0,C 180,E1 -5571.881,E2 -5571.881} C_VEL
LIN {X 0,Y 509.902,Z 396.943,A -85,B 0,C 180,E1 -5573.261,E2 -5573.261} C_VEL
LIN {X 0,Y 509.704,Z 401.958,A -85,B 0,C 180,E1 -5574.461,E2 -5574.461} C_VEL
LIN {X 0,Y 509.682,Z 405.771,A -85,B 0,C 180,E1 -5575.651,E2 -5575.651} C_VEL
LIN {X 0,Y 509.633,Z 408.572,A -85,B 0,C 180,E1 -5576.838,E2 -5576.838} C_VEL
LIN {X 0,Y 509.498,Z 409.934,A -85,B 0,C 180,E1 -5577.628,E2 -5577.628} C_VEL
LIN {X 0,Y 509.442,Z 411.423,A -85,B 0,C 180,E1 -5579.21,E2 -5579.21} C_VEL
LIN {X 0,Y 509.43,Z 411.603,A -85,B 0,C 180,E1 -5580,E2 -5580} C_VEL
LIN {X 0,Y 509.423,Z 411.38,A -85,B 0,C 180,E1 -5580.791,E2 -5580.791} C_VEL
LIN {X 0,Y 509.391,Z 409.749,A -85,B 0,C 180,E1 -5582.372,E2 -5582.372} C_VEL
LIN {X 0,Y 509.46,Z 408.346,A -85,B 0,C 180,E1 -5583.163,E2 -5583.163} C_VEL
LIN {X 0,Y 509.568,Z 405.419,A -85,B 0,C 180,E1 -5584.351,E2 -5584.351} C_VEL
LIN {X 0,Y 509.57,Z 401.501,A -85,B 0,C 180,E1 -5585.54,E2 -5585.54} C_VEL
LIN {X 0,Y 509.741,Z 396.627,A -85,B 0,C 180,E1 -5586.687,E2 -5586.687} C_VEL
LIN {X 0,Y 509.898,Z 390.105,A -85,B 0,C 180,E1 -5587.922,E2 -5587.922} C_VEL
LIN {X 0,Y 510.159,Z 382.176,A -85,B 0,C 180,E1 -5589.116,E2 -5589.116} C_VEL
LIN {X 0,Y 510.373,Z 374.112,A -85,B 0,C 180,E1 -5590.112,E2 -5590.112} C_VEL
LIN {X 0,Y 510.762,Z 364.276,A -85,B 0,C 180,E1 -5591.107,E2 -5591.107} C_VEL
LIN {X 0,Y 510.994,Z 354.67,A -85,B 0,C 180,E1 -5591.906,E2 -5591.906} C_VEL
LIN {X 0,Y 511.332,Z 342.651,A -85,B 0,C 180,E1 -5592.704,E2 -5592.704} C_VEL
LIN {X 0,Y 511.63,Z 329.93,A -85,B 0,C 180,E1 -5593.353,E2 -5593.353} C_VEL
LIN {X 0,Y 511.666,Z 317.269,A -85,B 0,C 180,E1 -5593.833,E2 -5593.833} C_VEL
LIN {X 0,Y 509.363,Z 307.342,A -85,B 0,C 180,E1 -5594.176,E2 -5594.176} C_VEL
LIN {X 0,Y 509.304,Z 304.459,A -85,B 0,C 180,E1 -5596.845,E2 -5596.845} C_VEL
LIN {X 0,Y 509.422,Z 300.877,A -85,B 0,C 180,E1 -5600.176,E2 -5600.176} C_VEL
LIN {X 0,Y 509.381,Z 298.153,A -85,B 0,C 180,E1 -5602.726,E2 -5602.726} C_VEL
LIN {X 0,Y 509.432,Z 295.394,A -85,B 0,C 180,E1 -5605.32,E2 -5605.32} C_VEL
LIN {X 0,Y 509.493,Z 292.5,A -85,B 0,C 180,E1 -5608.015,E2 -5608.015} C_VEL
LIN {X 0,Y 509.469,Z 289.071,A -85,B 0,C 180,E1 -5611.209,E2 -5611.209} C_VEL
LIN {X 0,Y 509.457,Z 287.654,A -85,B 0,C 180,E1 -5612.701,E2 -5612.701} C_VEL
LIN {X 0,Y 509.768,Z 287.615,A -85,B 0,C 180,E1 -5615.383,E2 -5615.383} C_VEL
LIN {X 0,Y 509.854,Z 287.598,A -85,B 0,C 180,E1 -5618.338,E2 -5618.338} C_VEL
LIN {X 0,Y 509.858,Z 287.596,A -85,B 0,C 180,E1 -5621.425,E2 -5621.425} C_VEL
LIN {X 0,Y 509.842,Z 287.602,A -85,B 0,C 180,E1 -5624.67,E2 -5624.67} C_VEL
LIN {X 0,Y 509.794,Z 287.608,A -85,B 0,C 180,E1 -5627.506,E2 -5627.506} C_VEL
LIN {X 0,Y 509.71,Z 287.622,A -85,B 0,C 180,E1 -5629.605,E2 -5629.605} C_VEL
LIN {X 0,Y 509.714,Z 287.89,A -85,B 0,C 180,E1 -5629.778,E2 -5629.778} C_VEL
LIN {X 0,Y 509.074,Z 288.993,A -85,B 0,C 180,E1 -5630.427,E2 -5630.427} C_VEL
LIN {X 0,Y 506.237,Z 290.954,A -85,B 0,C 180,E1 -5631.477,E2 -5631.477} C_VEL
LIN {X 0,Y 503.814,Z 292.515,A -85,B 0,C 180,E1 -5632.322,E2 -5632.322} C_VEL
LIN {X 0,Y 502.761,Z 293.601,A -85,B 0,C 180,E1 -5632.978,E2 -5632.978} C_VEL
LIN {X 0,Y 502.669,Z 293.936,A -85,B 0,C 180,E1 -5633.2,E2 -5633.2} C_VEL
LIN {X 0,Y 502.656,Z 297.863,A -85,B 0,C 180,E1 -5635.994,E2 -5635.994} C_VEL
LIN {X 0,Y 502.582,Z 301.723,A -85,B 0,C 180,E1 -5638.842,E2 -5638.842} C_VEL
LIN {X 0,Y 502.531,Z 305.649,A -85,B 0,C 180,E1 -5641.772,E2 -5641.772} C_VEL
LIN {X 0,Y 502.477,Z 309.158,A -85,B 0,C 180,E1 -5644.304,E2 -5644.304} C_VEL
LIN {X 0,Y 502.438,Z 313.683,A -85,B 0,C 180,E1 -5647.398,E2 -5647.398} C_VEL
LIN {X 0,Y 502.476,Z 317.478,A -85,B 0,C 180,E1 -5649.876,E2 -5649.876} C_VEL
LIN {X 0,Y 506.593,Z 331.006,A -85,B 0,C 180,E1 -5650.332,E2 -5650.332} C_VEL
LIN {X 0,Y 507.433,Z 335.354,A -85,B 0,C 180,E1 -5650.477,E2 -5650.477} C_VEL
LIN {X 0,Y 507.099,Z 350.077,A -85,B 0,C 180,E1 -5650.955,E2 -5650.955} C_VEL
LIN {X 0,Y 506.535,Z 364.835,A -85,B 0,C 180,E1 -5651.6,E2 -5651.6} C_VEL
LIN {X 0,Y 506.009,Z 379.189,A -85,B 0,C 180,E1 -5652.417,E2 -5652.417} C_VEL
LIN {X 0,Y 505.4,Z 392.183,A -85,B 0,C 180,E1 -5653.333,E2 -5653.333} C_VEL
LIN {X 0,Y 504.832,Z 403.425,A -85,B 0,C 180,E1 -5654.29,E2 -5654.29} C_VEL
LIN {X 0,Y 504.244,Z 415.074,A -85,B 0,C 180,E1 -5655.47,E2 -5655.47} C_VEL
LIN {X 0,Y 503.714,Z 425.171,A -85,B 0,C 180,E1 -5656.69,E2 -5656.69} C_VEL
LIN {X 0,Y 503.231,Z 434.704,A -85,B 0,C 180,E1 -5658.061,E2 -5658.061} C_VEL
LIN {X 0,Y 502.847,Z 443.212,A -85,B 0,C 180,E1 -5659.531,E2 -5659.531} C_VEL
LIN {X 0,Y 502.541,Z 450.865,A -85,B 0,C 180,E1 -5661.151,E2 -5661.151} C_VEL
LIN {X 0,Y 502.351,Z 456.948,A -85,B 0,C 180,E1 -5662.766,E2 -5662.766} C_VEL
LIN {X 0,Y 502.261,Z 461.648,A -85,B 0,C 180,E1 -5664.379,E2 -5664.379} C_VEL
LIN {X 0,Y 502.171,Z 465.1,A -85,B 0,C 180,E1 -5665.987,E2 -5665.987} C_VEL
LIN {X 0,Y 502.121,Z 467.378,A -85,B 0,C 180,E1 -5667.593,E2 -5667.593} C_VEL
LIN {X 0,Y 502.017,Z 468.546,A -85,B 0,C 180,E1 -5669.198,E2 -5669.198} C_VEL
LIN {X 0,Y 502.017,Z 468.563,A -85,B 0,C 180,E1 -5670.802,E2 -5670.802} C_VEL
LIN {X 0,Y 502.122,Z 467.46,A -85,B 0,C 180,E1 -5672.406,E2 -5672.406} C_VEL
LIN {X 0,Y 502.171,Z 465.252,A -85,B 0,C 180,E1 -5674.012,E2 -5674.012} C_VEL
LIN {X 0,Y 502.258,Z 461.88,A -85,B 0,C 180,E1 -5675.621,E2 -5675.621} C_VEL
LIN {X 0,Y 502.349,Z 457.258,A -85,B 0,C 180,E1 -5677.233,E2 -5677.233} C_VEL
LIN {X 0,Y 502.524,Z 451.251,A -85,B 0,C 180,E1 -5678.849,E2 -5678.849} C_VEL
LIN {X 0,Y 502.832,Z 443.685,A -85,B 0,C 180,E1 -5680.469,E2 -5680.469} C_VEL
LIN {X 0,Y 503.202,Z 435.306,A -85,B 0,C 180,E1 -5681.936,E2 -5681.936} C_VEL
LIN {X 0,Y 503.695,Z 425.862,A -85,B 0,C 180,E1 -5683.31,E2 -5683.31} C_VEL
LIN {X 0,Y 504.218,Z 415.901,A -85,B 0,C 180,E1 -5684.53,E2 -5684.53} C_VEL
LIN {X 0,Y 504.758,Z 404.635,A -85,B 0,C 180,E1 -5685.691,E2 -5685.691} C_VEL
LIN {X 0,Y 505.41,Z 392.274,A -85,B 0,C 180,E1 -5686.75,E2 -5686.75} C_VEL
LIN {X 0,Y 506.039,Z 378.969,A -85,B 0,C 180,E1 -5687.686,E2 -5687.686} C_VEL
LIN {X 0,Y 506.582,Z 364.544,A -85,B 0,C 180,E1 -5688.503,E2 -5688.503} C_VEL
LIN {X 0,Y 507.072,Z 349.439,A -85,B 0,C 180,E1 -5689.16,E2 -5689.16} C_VEL
LIN {X 0,Y 507.323,Z 334.012,A -85,B 0,C 180,E1 -5689.652,E2 -5689.652} C_VEL
LIN {X 0,Y 504.801,Z 324.838,A -85,B 0,C 180,E1 -5689.972,E2 -5689.972} C_VEL
LIN {X 0,Y 502.477,Z 317.443,A -85,B 0,C 180,E1 -5690.224,E2 -5690.224} C_VEL
LIN {X 0,Y 502.426,Z 313.138,A -85,B 0,C 180,E1 -5693.058,E2 -5693.058} C_VEL
LIN {X 0,Y 502.482,Z 309.303,A -85,B 0,C 180,E1 -5695.695,E2 -5695.695} C_VEL
LIN {X 0,Y 502.544,Z 305.558,A -85,B 0,C 180,E1 -5698.391,E2 -5698.391} C_VEL
LIN {X 0,Y 502.605,Z 301.455,A -85,B 0,C 180,E1 -5701.463,E2 -5701.463} C_VEL
LIN {X 0,Y 502.661,Z 297.449,A -85,B 0,C 180,E1 -5704.42,E2 -5704.42} C_VEL
LIN {X 0,Y 502.702,Z 293.574,A -85,B 0,C 180,E1 -5707.166,E2 -5707.166} C_VEL
LIN {X 0,Y 502.722,Z 289.711,A -85,B 0,C 180,E1 -5709.745,E2 -5709.745} C_VEL
LIN {X 0,Y 502.717,Z 288.497,A -85,B 0,C 180,E1 -5711.076,E2 -5711.076} C_VEL
LIN {X 0,Y 502.756,Z 288.488,A -85,B 0,C 180,E1 -5713.372,E2 -5713.372} C_VEL
LIN {X 0,Y 502.791,Z 288.483,A -85,B 0,C 180,E1 -5715.661,E2 -5715.661} C_VEL
LIN {X 0,Y 502.819,Z 288.478,A -85,B 0,C 180,E1 -5719.005,E2 -5719.005} C_VEL
LIN {X 0,Y 502.791,Z 288.484,A -85,B 0,C 180,E1 -5722.046,E2 -5722.046} C_VEL
LIN {X 0,Y 502.803,Z 288.481,A -85,B 0,C 180,E1 -5725.034,E2 -5725.034} C_VEL
LIN {X 0,Y 502.783,Z 288.48,A -85,B 0,C 180,E1 -5727.915,E2 -5727.915} C_VEL
LIN {X 0,Y 502.802,Z 288.478,A -85,B 0,C 180,E1 -5730.711,E2 -5730.711} C_VEL
LIN {X 0,Y 502.775,Z 288.482,A -85,B 0,C 180,E1 -5733.459,E2 -5733.459} C_VEL
LIN {X 0,Y 502.773,Z 288.481,A -85,B 0,C 180,E1 -5736.085,E2 -5736.085} C_VEL
LIN {X 0,Y 502.784,Z 288.479,A -85,B 0,C 180,E1 -5738.689,E2 -5738.689} C_VEL
LIN {X 0,Y 502.811,Z 288.476,A -85,B 0,C 180,E1 -5741.247,E2 -5741.247} C_VEL
LIN {X 0,Y 502.838,Z 288.471,A -85,B 0,C 180,E1 -5744.664,E2 -5744.664} C_VEL
LIN {X 0,Y 502.877,Z 288.464,A -85,B 0,C 180,E1 -5748.039,E2 -5748.039} C_VEL
LIN {X 0,Y 502.862,Z 288.47,A -85,B 0,C 180,E1 -5751.156,E2 -5751.156} C_VEL
LIN {X 0,Y 502.914,Z 288.457,A -85,B 0,C 180,E1 -5754.386,E2 -5754.386} C_VEL
LIN {X 0,Y 503.023,Z 288.449,A -85,B 0,C 180,E1 -5757.598,E2 -5757.598} C_VEL
LIN {X 0,Y 503.029,Z 288.444,A -85,B 0,C 180,E1 -5760,E2 -5760} C_VEL
LIN {X 0,Y 503.017,Z 288.451,A -85,B 0,C 180,E1 -5762.402,E2 -5762.402} C_VEL
LIN {X 0,Y 502.901,Z 288.462,A -85,B 0,C 180,E1 -5765.614,E2 -5765.614} C_VEL
LIN {X 0,Y 502.882,Z 288.468,A -85,B 0,C 180,E1 -5768.034,E2 -5768.034} C_VEL
LIN {X 0,Y 502.878,Z 288.46,A -85,B 0,C 180,E1 -5771.283,E2 -5771.283} C_VEL
LIN {X 0,Y 502.826,Z 288.474,A -85,B 0,C 180,E1 -5774.571,E2 -5774.571} C_VEL
LIN {X 0,Y 502.822,Z 288.473,A -85,B 0,C 180,E1 -5777.908,E2 -5777.908} C_VEL
LIN {X 0,Y 502.829,Z 288.472,A -85,B 0,C 180,E1 -5780.536,E2 -5780.536} C_VEL
LIN {X 0,Y 502.787,Z 288.478,A -85,B 0,C 180,E1 -5783.041,E2 -5783.041} C_VEL
LIN {X 0,Y 502.778,Z 288.477,A -85,B 0,C 180,E1 -5785.679,E2 -5785.679} C_VEL
LIN {X 0,Y 502.795,Z 288.48,A -85,B 0,C 180,E1 -5788.375,E2 -5788.375} C_VEL
LIN {X 0,Y 502.796,Z 288.478,A -85,B 0,C 180,E1 -5791.143,E2 -5791.143} C_VEL
LIN {X 0,Y 502.803,Z 288.478,A -85,B 0,C 180,E1 -5793.994,E2 -5793.994} C_VEL
LIN {X 0,Y 502.763,Z 288.485,A -85,B 0,C 180,E1 -5797.176,E2 -5797.176} C_VEL
LIN {X 0,Y 502.784,Z 288.483,A -85,B 0,C 180,E1 -5800.015,E2 -5800.015} C_VEL
LIN {X 0,Y 502.802,Z 288.478,A -85,B 0,C 180,E1 -5802.199,E2 -5802.199} C_VEL
LIN {X 0,Y 502.785,Z 288.479,A -85,B 0,C 180,E1 -5805.47,E2 -5805.47} C_VEL
LIN {X 0,Y 502.794,Z 288.476,A -85,B 0,C 180,E1 -5807.861,E2 -5807.861} C_VEL
LIN {X 0,Y 502.808,Z 288.584,A -85,B 0,C 180,E1 -5809.987,E2 -5809.987} C_VEL
LIN {X 0,Y 506.17,Z 301.667,A -85,B 0,C 180,E1 -5813.094,E2 -5813.094} C_VEL
LIN {X 0,Y 507.947,Z 308.89,A -85,B 0,C 180,E1 -5814.719,E2 -5814.719} C_VEL
LIN {X 0,Y 507.608,Z 316.284,A -85,B 0,C 180,E1 -5816.173,E2 -5816.173} C_VEL
LIN {X 0,Y 506.601,Z 330.664,A -85,B 0,C 180,E1 -5818.885,E2 -5818.885} C_VEL
LIN {X 0,Y 505.784,Z 345.601,A -85,B 0,C 180,E1 -5821.603,E2 -5821.603} C_VEL
LIN {X 0,Y 504.926,Z 363.734,A -85,B 0,C 180,E1 -5824.786,E2 -5824.786} C_VEL
LIN {X 0,Y 504.229,Z 382.021,A -85,B 0,C 180,E1 -5827.894,E2 -5827.894} C_VEL
LIN {X 0,Y 503.836,Z 394.471,A -85,B 0,C 180,E1 -5829.963,E2 -5829.963} C_VEL
LIN {X 0,Y 506.196,Z 408.582,A -85,B 0,C 180,E1 -5830.279,E2 -5830.279} C_VEL
LIN {X 0,Y 506.902,Z 413.296,A -85,B 0,C 180,E1 -5830.406,E2 -5830.406} C_VEL
LIN {X 0,Y 506.512,Z 428.351,A -85,B 0,C 180,E1 -5830.822,E2 -5830.822} C_VEL
LIN {X 0,Y 506.041,Z 443.872,A -85,B 0,C 180,E1 -5831.424,E2 -5831.424} C_VEL
LIN {X 0,Y 505.467,Z 458.886,A -85,B 0,C 180,E1 -5832.189,E2 -5832.189} C_VEL
LIN {X 0,Y 504.952,Z 471.751,A -85,B 0,C 180,E1 -5833.006,E2 -5833.006} C_VEL
LIN {X 0,Y 504.399,Z 485.044,A -85,B 0,C 180,E1 -5834.03,E2 -5834.03} C_VEL
LIN {X 0,Y 503.853,Z 497.155,A -85,B 0,C 180,E1 -5835.149,E2 -5835.149} C_VEL
LIN {X 0,Y 503.386,Z 509.122,A -85,B 0,C 180,E1 -5836.476,E2 -5836.476} C_VEL
LIN {X 0,Y 502.943,Z 519.81,A -85,B 0,C 180,E1 -5837.901,E2 -5837.901} C_VEL
LIN {X 0,Y 502.741,Z 528.719,A -85,B 0,C 180,E1 -5839.326,E2 -5839.326} C_VEL
LIN {X 0,Y 502.447,Z 536.108,A -85,B 0,C 180,E1 -5840.744,E2 -5840.744} C_VEL
LIN {X 0,Y 502.295,Z 542.97,A -85,B 0,C 180,E1 -5842.362,E2 -5842.362} C_VEL
LIN {X 0,Y 502.202,Z 547.797,A -85,B 0,C 180,E1 -5843.785,E2 -5843.785} C_VEL
LIN {X 0,Y 502.098,Z 551.436,A -85,B 0,C 180,E1 -5845.183,E2 -5845.183} C_VEL
LIN {X 0,Y 502.138,Z 554.475,A -85,B 0,C 180,E1 -5846.791,E2 -5846.791} C_VEL
LIN {X 0,Y 502.038,Z 556.268,A -85,B 0,C 180,E1 -5848.396,E2 -5848.396} C_VEL
LIN {X 0,Y 501.991,Z 556.875,A -85,B 0,C 180,E1 -5850,E2 -5850} C_VEL
LIN {X 0,Y 502.039,Z 556.256,A -85,B 0,C 180,E1 -5851.605,E2 -5851.605} C_VEL
LIN {X 0,Y 502.138,Z 554.445,A -85,B 0,C 180,E1 -5853.21,E2 -5853.21} C_VEL
LIN {X 0,Y 502.115,Z 551.388,A -85,B 0,C 180,E1 -5854.818,E2 -5854.818} C_VEL
LIN {X 0,Y 502.273,Z 547.05,A -85,B 0,C 180,E1 -5856.427,E2 -5856.427} C_VEL
LIN {X 0,Y 502.324,Z 541.269,A -85,B 0,C 180,E1 -5858.043,E2 -5858.043} C_VEL
LIN {X 0,Y 502.447,Z 535.905,A -85,B 0,C 180,E1 -5859.257,E2 -5859.257} C_VEL
LIN {X 0,Y 502.74,Z 528.432,A -85,B 0,C 180,E1 -5860.675,E2 -5860.675} C_VEL
LIN {X 0,Y 502.94,Z 519.406,A -85,B 0,C 180,E1 -5862.1,E2 -5862.1} C_VEL
LIN {X 0,Y 503.386,Z 508.558,A -85,B 0,C 180,E1 -5863.524,E2 -5863.524} C_VEL
LIN {X 0,Y 503.776,Z 497.41,A -85,B 0,C 180,E1 -5864.75,E2 -5864.75} C_VEL
LIN {X 0,Y 504.339,Z 484.382,A -85,B 0,C 180,E1 -5865.947,E2 -5865.947} C_VEL
LIN {X 0,Y 504.89,Z 470.516,A -85,B 0,C 180,E1 -5866.997,E2 -5866.997} C_VEL
LIN {X 0,Y 505.412,Z 457.373,A -85,B 0,C 180,E1 -5867.814,E2 -5867.814} C_VEL
LIN {X 0,Y 505.955,Z 443.174,A -85,B 0,C 180,E1 -5868.527,E2 -5868.527} C_VEL
LIN {X 0,Y 506.363,Z 427.291,A -85,B 0,C 180,E1 -5869.142,E2 -5869.142} C_VEL
LIN {X 0,Y 506.722,Z 412.107,A -85,B 0,C 180,E1 -5869.559,E2 -5869.559} C_VEL
LIN {X 0,Y 504.368,Z 398.753,A -85,B 0,C 180,E1 -5869.884,E2 -5869.884} C_VEL
LIN {X 0,Y 503.705,Z 393.11,A -85,B 0,C 180,E1 -5870.016,E2 -5870.016} C_VEL
LIN {X 0,Y 504.145,Z 374.691,A -85,B 0,C 180,E1 -5872.975,E2 -5872.975} C_VEL
LIN {X 0,Y 504.652,Z 357.878,A -85,B 0,C 180,E1 -5875.798,E2 -5875.798} C_VEL
LIN {X 0,Y 505.407,Z 342.557,A -85,B 0,C 180,E1 -5878.537,E2 -5878.537} C_VEL
LIN {X 0,Y 506.178,Z 330.221,A -85,B 0,C 180,E1 -5880.912,E2 -5880.912} C_VEL
LIN {X 0,Y 507.579,Z 317.482,A -85,B 0,C 180,E1 -5883.631,E2 -5883.631} C_VEL
LIN {X 0,Y 508.348,Z 311.946,A -85,B 0,C 180,E1 -5884.935,E2 -5884.935} C_VEL
LIN {X 0,Y 508.291,Z 309.846,A -85,B 0,C 180,E1 -5885.502,E2 -5885.502} C_VEL
LIN {X 0,Y 507.011,Z 304.874,A -85,B 0,C 180,E1 -5887.084,E2 -5887.084} C_VEL
LIN {X 0,Y 505.774,Z 300.069,A -85,B 0,C 180,E1 -5888.909,E2 -5888.909} C_VEL
LIN {X 0,Y 504.591,Z 295.528,A -85,B 0,C 180,E1 -5891.226,E2 -5891.226} C_VEL
LIN {X 0,Y 503.791,Z 292.662,A -85,B 0,C 180,E1 -5893.497,E2 -5893.497} C_VEL
LIN {X 0,Y 503.464,Z 291.195,A -85,B 0,C 180,E1 -5895.736,E2 -5895.736} C_VEL
LIN {X 0,Y 503.374,Z 290.908,A -85,B 0,C 180,E1 -5897.92,E2 -5897.92} C_VEL
LIN {X 0,Y 503.4,Z 291.494,A -85,B 0,C 180,E1 -5900.162,E2 -5900.162} C_VEL
LIN {X 0,Y 503.559,Z 293.081,A -85,B 0,C 180,E1 -5903.12,E2 -5903.12} C_VEL
LIN {X 0,Y 503.528,Z 295.19,A -85,B 0,C 180,E1 -5906.062,E2 -5906.062} C_VEL
LIN {X 0,Y 503.327,Z 297.413,A -85,B 0,C 180,E1 -5908.893,E2 -5908.893} C_VEL
LIN {X 0,Y 503.269,Z 299.637,A -85,B 0,C 180,E1 -5911.654,E2 -5911.654} C_VEL
LIN {X 0,Y 503.136,Z 301.733,A -85,B 0,C 180,E1 -5914.341,E2 -5914.341} C_VEL
LIN {X 0,Y 503.031,Z 304.063,A -85,B 0,C 180,E1 -5917.237,E2 -5917.237} C_VEL
LIN {X 0,Y 502.892,Z 306.693,A -85,B 0,C 180,E1 -5920.403,E2 -5920.403} C_VEL
LIN {X 0,Y 502.804,Z 308.855,A -85,B 0,C 180,E1 -5922.931,E2 -5922.931} C_VEL
LIN {X 0,Y 502.754,Z 311.362,A -85,B 0,C 180,E1 -5925.582,E2 -5925.582} C_VEL
LIN {X 0,Y 505.508,Z 319.971,A -85,B 0,C 180,E1 -5925.944,E2 -5925.944} C_VEL
LIN {X 0,Y 505.242,Z 332.26,A -85,B 0,C 180,E1 -5926.424,E2 -5926.424} C_VEL
LIN {X 0,Y 504.922,Z 343.985,A -85,B 0,C 180,E1 -5927.04,E2 -5927.04} C_VEL
LIN {X 0,Y 504.497,Z 356.166,A -85,B 0,C 180,E1 -5927.862,E2 -5927.862} C_VEL
LIN {X 0,Y 504.155,Z 366.573,A -85,B 0,C 180,E1 -5928.746,E2 -5928.746} C_VEL
LIN {X 0,Y 503.789,Z 376.173,A -85,B 0,C 180,E1 -5929.755,E2 -5929.755} C_VEL
LIN {X 0,Y 503.423,Z 385.52,A -85,B 0,C 180,E1 -5930.964,E2 -5930.964} C_VEL
LIN {X 0,Y 503.136,Z 393.112,A -85,B 0,C 180,E1 -5932.193,E2 -5932.193} C_VEL
LIN {X 0,Y 502.937,Z 399.848,A -85,B 0,C 180,E1 -5933.581,E2 -5933.581} C_VEL
LIN {X 0,Y 502.687,Z 404.42,A -85,B 0,C 180,E1 -5934.786,E2 -5934.786} C_VEL
LIN {X 0,Y 502.59,Z 407.887,A -85,B 0,C 180,E1 -5935.991,E2 -5935.991} C_VEL
LIN {X 0,Y 502.638,Z 409.646,A -85,B 0,C 180,E1 -5936.794,E2 -5936.794} C_VEL
LIN {X 0,Y 502.497,Z 410.999,A -85,B 0,C 180,E1 -5937.595,E2 -5937.595} C_VEL
LIN {X 0,Y 502.386,Z 411.936,A -85,B 0,C 180,E1 -5938.397,E2 -5938.397} C_VEL
LIN {X 0,Y 502.436,Z 412.471,A -85,B 0,C 180,E1 -5939.199,E2 -5939.199} C_VEL
LIN {X 0,Y 502.423,Z 412.637,A -85,B 0,C 180,E1 -5940,E2 -5940} C_VEL
LIN {X 0,Y 502.418,Z 412.398,A -85,B 0,C 180,E1 -5940.802,E2 -5940.802} C_VEL
LIN {X 0,Y 502.368,Z 410.742,A -85,B 0,C 180,E1 -5942.405,E2 -5942.405} C_VEL
LIN {X 0,Y 502.438,Z 409.321,A -85,B 0,C 180,E1 -5943.208,E2 -5943.208} C_VEL
LIN {X 0,Y 502.558,Z 406.369,A -85,B 0,C 180,E1 -5944.411,E2 -5944.411} C_VEL
LIN {X 0,Y 502.57,Z 402.421,A -85,B 0,C 180,E1 -5945.618,E2 -5945.618} C_VEL
LIN {X 0,Y 502.753,Z 397.926,A -85,B 0,C 180,E1 -5946.693,E2 -5946.693} C_VEL
LIN {X 0,Y 502.928,Z 390.96,A -85,B 0,C 180,E1 -5948.033,E2 -5948.033} C_VEL
LIN {X 0,Y 503.207,Z 382.997,A -85,B 0,C 180,E1 -5949.243,E2 -5949.243} C_VEL
LIN {X 0,Y 503.442,Z 374.91,A -85,B 0,C 180,E1 -5950.253,E2 -5950.253} C_VEL
LIN {X 0,Y 503.855,Z 365.055,A -85,B 0,C 180,E1 -5951.261,E2 -5951.261} C_VEL
LIN {X 0,Y 504.107,Z 355.438,A -85,B 0,C 180,E1 -5952.071,E2 -5952.071} C_VEL
LIN {X 0,Y 504.478,Z 343.432,A -85,B 0,C 180,E1 -5952.88,E2 -5952.88} C_VEL
LIN {X 0,Y 504.785,Z 330.756,A -85,B 0,C 180,E1 -5953.537,E2 -5953.537} C_VEL
LIN {X 0,Y 504.853,Z 318.251,A -85,B 0,C 180,E1 -5954.023,E2 -5954.023} C_VEL
LIN {X 0,Y 502.316,Z 307.851,A -85,B 0,C 180,E1 -5954.405,E2 -5954.405} C_VEL
LIN {X 0,Y 502.296,Z 304.024,A -85,B 0,C 180,E1 -5957.928,E2 -5957.928} C_VEL
LIN {X 0,Y 502.322,Z 301.281,A -85,B 0,C 180,E1 -5960.474,E2 -5960.474} C_VEL
LIN {X 0,Y 502.322,Z 298.519,A -85,B 0,C 180,E1 -5963.063,E2 -5963.063} C_VEL
LIN {X 0,Y 502.35,Z 295.712,A -85,B 0,C 180,E1 -5965.703,E2 -5965.703} C_VEL
LIN {X 0,Y 502.416,Z 292.809,A -85,B 0,C 180,E1 -5968.399,E2 -5968.399} C_VEL
LIN {X 0,Y 502.405,Z 289.548,A -85,B 0,C 180,E1 -5971.426,E2 -5971.426} C_VEL
LIN {X 0,Y 502.394,Z 288.825,A -85,B 0,C 180,E1 -5972.113,E2 -5972.113} C_VEL
LIN {X 0,Y 502.652,Z 288.499,A -85,B 0,C 180,E1 -5974.418,E2 -5974.418} C_VEL
LIN {X 0,Y 502.765,Z 288.487,A -85,B 0,C 180,E1 -5977.175,E2 -5977.175} C_VEL
LIN {X 0,Y 502.791,Z 288.477,A -85,B 0,C 180,E1 -5980.015,E2 -5980.015} C_VEL
LIN {X 0,Y 502.806,Z 288.476,A -85,B 0,C 180,E1 -5982.199,E2 -5982.199} C_VEL
LIN {X 0,Y 502.788,Z 288.478,A -85,B 0,C 180,E1 -5985.47,E2 -5985.47} C_VEL
LIN {X 0,Y 502.767,Z 288.487,A -85,B 0,C 180,E1 -5987.857,E2 -5987.857} C_VEL
LIN {X 0,Y 502.679,Z 288.512,A -85,B 0,C 180,E1 -5989.581,E2 -5989.581} C_VEL
LIN {X 0,Y 502.735,Z 292.246,A -85,B 0,C 180,E1 -5992.041,E2 -5992.041} C_VEL
LIN {X 0,Y 502.669,Z 293.936,A -85,B 0,C 180,E1 -5993.2,E2 -5993.2} C_VEL
LIN {X 0,Y 501.983,Z 294.993,A -85,B 0,C 180,E1 -5993.859,E2 -5993.859} C_VEL
LIN {X 0,Y 499.114,Z 296.85,A -85,B 0,C 180,E1 -5994.925,E2 -5994.925} C_VEL
LIN {X 0,Y 496.703,Z 298.34,A -85,B 0,C 180,E1 -5995.784,E2 -5995.784} C_VEL
LIN {X 0,Y 495.675,Z 299.367,A -85,B 0,C 180,E1 -5996.45,E2 -5996.45} C_VEL
LIN {X 0,Y 495.595,Z 299.681,A -85,B 0,C 180,E1 -5996.676,E2 -5996.676} C_VEL
LIN {X 0,Y 495.507,Z 303.223,A -85,B 0,C 180,E1 -5999.296,E2 -5999.296} C_VEL
LIN {X 0,Y 495.461,Z 306.981,A -85,B 0,C 180,E1 -6002.089,E2 -6002.089} C_VEL
LIN {X 0,Y 495.425,Z 310.774,A -85,B 0,C 180,E1 -6004.813,E2 -6004.813} C_VEL
LIN {X 0,Y 495.41,Z 314.702,A -85,B 0,C 180,E1 -6007.478,E2 -6007.478} C_VEL
LIN {X 0,Y 495.443,Z 318.03,A -85,B 0,C 180,E1 -6009.589,E2 -6009.589} C_VEL
LIN {X 0,Y 499.992,Z 332.402,A -85,B 0,C 180,E1 -6010.082,E2 -6010.082} C_VEL
LIN {X 0,Y 500.738,Z 336.946,A -85,B 0,C 180,E1 -6010.235,E2 -6010.235} C_VEL
LIN {X 0,Y 500.409,Z 351.152,A -85,B 0,C 180,E1 -6010.709,E2 -6010.709} C_VEL
LIN {X 0,Y 499.825,Z 365.429,A -85,B 0,C 180,E1 -6011.344,E2 -6011.344} C_VEL
LIN {X 0,Y 499.279,Z 379.787,A -85,B 0,C 180,E1 -6012.172,E2 -6012.172} C_VEL
LIN {X 0,Y 498.631,Z 392.784,A -85,B 0,C 180,E1 -6013.1,E2 -6013.1} C_VEL
LIN {X 0,Y 498.021,Z 404.193,A -85,B 0,C 180,E1 -6014.085,E2 -6014.085} C_VEL
LIN {X 0,Y 497.405,Z 415.677,A -85,B 0,C 180,E1 -6015.266,E2 -6015.266} C_VEL
LIN {X 0,Y 496.839,Z 425.774,A -85,B 0,C 180,E1 -6016.502,E2 -6016.502} C_VEL
LIN {X 0,Y 496.281,Z 435.504,A -85,B 0,C 180,E1 -6017.921,E2 -6017.921} C_VEL
LIN {X 0,Y 495.878,Z 443.819,A -85,B 0,C 180,E1 -6019.383,E2 -6019.383} C_VEL
LIN {X 0,Y 495.536,Z 451.474,A -85,B 0,C 180,E1 -6021.024,E2 -6021.024} C_VEL
LIN {X 0,Y 495.331,Z 457.556,A -85,B 0,C 180,E1 -6022.663,E2 -6022.663} C_VEL
LIN {X 0,Y 495.206,Z 462.258,A -85,B 0,C 180,E1 -6024.298,E2 -6024.298} C_VEL
LIN {X 0,Y 495.109,Z 465.709,A -85,B 0,C 180,E1 -6025.93,E2 -6025.93} C_VEL
LIN {X 0,Y 495.056,Z 467.986,A -85,B 0,C 180,E1 -6027.559,E2 -6027.559} C_VEL
LIN {X 0,Y 494.944,Z 469.154,A -85,B 0,C 180,E1 -6029.186,E2 -6029.186} C_VEL
LIN {X 0,Y 494.944,Z 469.171,A -85,B 0,C 180,E1 -6030.813,E2 -6030.813} C_VEL
LIN {X 0,Y 495.057,Z 468.068,A -85,B 0,C 180,E1 -6032.441,E2 -6032.441} C_VEL
LIN {X 0,Y 495.109,Z 465.859,A -85,B 0,C 180,E1 -6034.07,E2 -6034.07} C_VEL
LIN {X 0,Y 495.201,Z 462.487,A -85,B 0,C 180,E1 -6035.701,E2 -6035.701} C_VEL
LIN {X 0,Y 495.33,Z 457.862,A -85,B 0,C 180,E1 -6037.336,E2 -6037.336} C_VEL
LIN {X 0,Y 495.518,Z 451.855,A -85,B 0,C 180,E1 -6038.975,E2 -6038.975} C_VEL
LIN {X 0,Y 495.862,Z 444.286,A -85,B 0,C 180,E1 -6040.617,E2 -6040.617} C_VEL
LIN {X 0,Y 496.262,Z 436.215,A -85,B 0,C 180,E1 -6042.056,E2 -6042.056} C_VEL
LIN {X 0,Y 496.79,Z 426.459,A -85,B 0,C 180,E1 -6043.498,E2 -6043.498} C_VEL
LIN {X 0,Y 497.372,Z 416.493,A -85,B 0,C 180,E1 -6044.735,E2 -6044.735} C_VEL
LIN {X 0,Y 497.943,Z 405.368,A -85,B 0,C 180,E1 -6045.898,E2 -6045.898} C_VEL
LIN {X 0,Y 498.651,Z 392.857,A -85,B 0,C 180,E1 -6046.983,E2 -6046.983} C_VEL
LIN {X 0,Y 499.305,Z 379.547,A -85,B 0,C 180,E1 -6047.933,E2 -6047.933} C_VEL
LIN {X 0,Y 499.89,Z 365.11,A -85,B 0,C 180,E1 -6048.76,E2 -6048.76} C_VEL
LIN {X 0,Y 500.398,Z 349.869,A -85,B 0,C 180,E1 -6049.431,E2 -6049.431} C_VEL
LIN {X 0,Y 500.642,Z 335.272,A -85,B 0,C 180,E1 -6049.907,E2 -6049.907} C_VEL
LIN {X 0,Y 498.161,Z 326.492,A -85,B 0,C 180,E1 -6050.226,E2 -6050.226} C_VEL
LIN {X 0,Y 495.437,Z 317.939,A -85,B 0,C 180,E1 -6050.524,E2 -6050.524} C_VEL
LIN {X 0,Y 495.373,Z 313.517,A -85,B 0,C 180,E1 -6053.406,E2 -6053.406} C_VEL
LIN {X 0,Y 495.44,Z 309.65,A -85,B 0,C 180,E1 -6056.088,E2 -6056.088} C_VEL
LIN {X 0,Y 495.492,Z 305.855,A -85,B 0,C 180,E1 -6058.832,E2 -6058.832} C_VEL
LIN {X 0,Y 495.572,Z 302.047,A -85,B 0,C 180,E1 -6061.691,E2 -6061.691} C_VEL
LIN {X 0,Y 495.612,Z 298.011,A -85,B 0,C 180,E1 -6064.667,E2 -6064.667} C_VEL
LIN {X 0,Y 495.683,Z 293.915,A -85,B 0,C 180,E1 -6067.566,E2 -6067.566} C_VEL
LIN {X 0,Y 495.675,Z 290.228,A -85,B 0,C 180,E1 -6070.035,E2 -6070.035} C_VEL
LIN {X 0,Y 495.626,Z 289.382,A -85,B 0,C 180,E1 -6070.714,E2 -6070.714} C_VEL
LIN {X 0,Y 495.699,Z 289.364,A -85,B 0,C 180,E1 -6072.886,E2 -6072.886} C_VEL
LIN {X 0,Y 495.734,Z 289.36,A -85,B 0,C 180,E1 -6075.999,E2 -6075.999} C_VEL
LIN {X 0,Y 495.765,Z 289.354,A -85,B 0,C 180,E1 -6079.3,E2 -6079.3} C_VEL
LIN {X 0,Y 495.727,Z 289.36,A -85,B 0,C 180,E1 -6082.438,E2 -6082.438} C_VEL
LIN {X 0,Y 495.782,Z 289.354,A -85,B 0,C 180,E1 -6085.457,E2 -6085.457} C_VEL
LIN {X 0,Y 495.755,Z 289.358,A -85,B 0,C 180,E1 -6088.364,E2 -6088.364} C_VEL
LIN {X 0,Y 495.724,Z 289.358,A -85,B 0,C 180,E1 -6091.182,E2 -6091.182} C_VEL
LIN {X 0,Y 495.723,Z 289.358,A -85,B 0,C 180,E1 -6093.928,E2 -6093.928} C_VEL
LIN {X 0,Y 495.76,Z 289.354,A -85,B 0,C 180,E1 -6097.139,E2 -6097.139} C_VEL
LIN {X 0,Y 495.768,Z 289.356,A -85,B 0,C 180,E1 -6100.109,E2 -6100.109} C_VEL
LIN {X 0,Y 495.742,Z 289.351,A -85,B 0,C 180,E1 -6102.68,E2 -6102.68} C_VEL
LIN {X 0,Y 495.795,Z 289.354,A -85,B 0,C 180,E1 -6105.217,E2 -6105.217} C_VEL
LIN {X 0,Y 495.852,Z 289.34,A -85,B 0,C 180,E1 -6108.555,E2 -6108.555} C_VEL
LIN {X 0,Y 495.82,Z 289.352,A -85,B 0,C 180,E1 -6111.851,E2 -6111.851} C_VEL
LIN {X 0,Y 495.829,Z 289.344,A -85,B 0,C 180,E1 -6115.121,E2 -6115.121} C_VEL
LIN {X 0,Y 495.992,Z 289.325,A -85,B 0,C 180,E1 -6117.564,E2 -6117.564} C_VEL
LIN {X 0,Y 496,Z 289.319,A -85,B 0,C 180,E1 -6120,E2 -6120} C_VEL
LIN {X 0,Y 495.985,Z 289.327,A -85,B 0,C 180,E1 -6122.436,E2 -6122.436} C_VEL
LIN {X 0,Y 495.861,Z 289.338,A -85,B 0,C 180,E1 -6125.694,E2 -6125.694} C_VEL
LIN {X 0,Y 495.838,Z 289.346,A -85,B 0,C 180,E1 -6128.148,E2 -6128.148} C_VEL
LIN {X 0,Y 495.852,Z 289.336,A -85,B 0,C 180,E1 -6131.445,E2 -6131.445} C_VEL
LIN {X 0,Y 495.777,Z 289.353,A -85,B 0,C 180,E1 -6134.783,E2 -6134.783} C_VEL
LIN {X 0,Y 495.759,Z 289.354,A -85,B 0,C 180,E1 -6137.319,E2 -6137.319} C_VEL
LIN {X 0,Y 495.772,Z 289.355,A -85,B 0,C 180,E1 -6139.89,E2 -6139.89} C_VEL
LIN {X 0,Y 495.758,Z 289.352,A -85,B 0,C 180,E1 -6142.86,E2 -6142.86} C_VEL
LIN {X 0,Y 495.721,Z 289.355,A -85,B 0,C 180,E1 -6146.072,E2 -6146.072} C_VEL
LIN {X 0,Y 495.743,Z 289.359,A -85,B 0,C 180,E1 -6148.816,E2 -6148.816} C_VEL
LIN {X 0,Y 495.755,Z 289.359,A -85,B 0,C 180,E1 -6151.725,E2 -6151.725} C_VEL
LIN {X 0,Y 495.767,Z 289.354,A -85,B 0,C 180,E1 -6154.694,E2 -6154.694} C_VEL
LIN {X 0,Y 495.719,Z 289.36,A -85,B 0,C 180,E1 -6157.562,E2 -6157.562} C_VEL
LIN {X 0,Y 495.765,Z 289.354,A -85,B 0,C 180,E1 -6160.7,E2 -6160.7} C_VEL
LIN {X 0,Y 495.727,Z 289.358,A -85,B 0,C 180,E1 -6164.002,E2 -6164.002} C_VEL
LIN {X 0,Y 495.705,Z 289.362,A -85,B 0,C 180,E1 -6167.115,E2 -6167.115} C_VEL
LIN {X 0,Y 495.763,Z 289.467,A -85,B 0,C 180,E1 -6169.526,E2 -6169.526} C_VEL
LIN {X 0,Y 499.199,Z 302.682,A -85,B 0,C 180,E1 -6172.744,E2 -6172.744} C_VEL
LIN {X 0,Y 501.183,Z 310.891,A -85,B 0,C 180,E1 -6174.614,E2 -6174.614} C_VEL
LIN {X 0,Y 500.715,Z 319.502,A -85,B 0,C 180,E1 -6176.329,E2 -6176.329} C_VEL
LIN {X 0,Y 499.602,Z 334.629,A -85,B 0,C 180,E1 -6179.219,E2 -6179.219} C_VEL
LIN {X 0,Y 498.816,Z 347.551,A -85,B 0,C 180,E1 -6181.607,E2 -6181.607} C_VEL
LIN {X 0,Y 497.964,Z 364.217,A -85,B 0,C 180,E1 -6184.59,E2 -6184.59} C_VEL
LIN {X 0,Y 497.267,Z 381.385,A -85,B 0,C 180,E1 -6187.567,E2 -6187.567} C_VEL
LIN {X 0,Y 496.887,Z 393.995,A -85,B 0,C 180,E1 -6189.711,E2 -6189.711} C_VEL
LIN {X 0,Y 499.224,Z 408.778,A -85,B 0,C 180,E1 -6190.047,E2 -6190.047} C_VEL
LIN {X 0,Y 500.077,Z 414.367,A -85,B 0,C 180,E1 -6190.205,E2 -6190.205} C_VEL
LIN {X 0,Y 499.637,Z 429.491,A -85,B 0,C 180,E1 -6190.649,E2 -6190.649} C_VEL
LIN {X 0,Y 499.124,Z 444.621,A -85,B 0,C 180,E1 -6191.264,E2 -6191.264} C_VEL
LIN {X 0,Y 498.522,Z 459.295,A -85,B 0,C 180,E1 -6192.038,E2 -6192.038} C_VEL
LIN {X 0,Y 497.914,Z 473.37,A -85,B 0,C 180,E1 -6192.969,E2 -6192.969} C_VEL
LIN {X 0,Y 497.343,Z 486.686,A -85,B 0,C 180,E1 -6194.047,E2 -6194.047} C_VEL
LIN {X 0,Y 496.793,Z 498.01,A -85,B 0,C 180,E1 -6195.143,E2 -6195.143} C_VEL
LIN {X 0,Y 496.28,Z 509.691,A -85,B 0,C 180,E1 -6196.487,E2 -6196.487} C_VEL
LIN {X 0,Y 495.905,Z 518.748,A -85,B 0,C 180,E1 -6197.727,E2 -6197.727} C_VEL
LIN {X 0,Y 495.691,Z 527.689,A -85,B 0,C 180,E1 -6199.172,E2 -6199.172} C_VEL
LIN {X 0,Y 495.361,Z 535.099,A -85,B 0,C 180,E1 -6200.61,E2 -6200.61} C_VEL
LIN {X 0,Y 495.234,Z 541.983,A -85,B 0,C 180,E1 -6202.252,E2 -6202.252} C_VEL
LIN {X 0,Y 495.161,Z 547.063,A -85,B 0,C 180,E1 -6203.778,E2 -6203.778} C_VEL
LIN {X 0,Y 495.077,Z 550.469,A -85,B 0,C 180,E1 -6205.114,E2 -6205.114} C_VEL
LIN {X 0,Y 495.089,Z 553.505,A -85,B 0,C 180,E1 -6206.745,E2 -6206.745} C_VEL
LIN {X 0,Y 495.002,Z 555.295,A -85,B 0,C 180,E1 -6208.373,E2 -6208.373} C_VEL
LIN {X 0,Y 494.96,Z 555.891,A -85,B 0,C 180,E1 -6210,E2 -6210} C_VEL
LIN {X 0,Y 495.007,Z 555.257,A -85,B 0,C 180,E1 -6211.627,E2 -6211.627} C_VEL
LIN {X 0,Y 495.095,Z 553.428,A -85,B 0,C 180,E1 -6213.255,E2 -6213.255} C_VEL
LIN {X 0,Y 495.092,Z 550.344,A -85,B 0,C 180,E1 -6214.886,E2 -6214.886} C_VEL
LIN {X 0,Y 495.232,Z 545.741,A -85,B 0,C 180,E1 -6216.59,E2 -6216.59} C_VEL
LIN {X 0,Y 495.276,Z 540.14,A -85,B 0,C 180,E1 -6218.158,E2 -6218.158} C_VEL
LIN {X 0,Y 495.418,Z 532.729,A -85,B 0,C 180,E1 -6219.802,E2 -6219.802} C_VEL
LIN {X 0,Y 495.733,Z 524.81,A -85,B 0,C 180,E1 -6221.241,E2 -6221.241} C_VEL
LIN {X 0,Y 496.014,Z 515.244,A -85,B 0,C 180,E1 -6222.687,E2 -6222.687} C_VEL
LIN {X 0,Y 496.423,Z 505.484,A -85,B 0,C 180,E1 -6223.927,E2 -6223.927} C_VEL
LIN {X 0,Y 496.891,Z 492.879,A -85,B 0,C 180,E1 -6225.274,E2 -6225.274} C_VEL
LIN {X 0,Y 497.526,Z 480.098,A -85,B 0,C 180,E1 -6226.411,E2 -6226.411} C_VEL
LIN {X 0,Y 498.039,Z 467.671,A -85,B 0,C 180,E1 -6227.344,E2 -6227.344} C_VEL
LIN {X 0,Y 498.565,Z 454.218,A -85,B 0,C 180,E1 -6228.173,E2 -6228.173} C_VEL
LIN {X 0,Y 499.168,Z 439.418,A -85,B 0,C 180,E1 -6228.895,E2 -6228.895} C_VEL
LIN {X 0,Y 499.61,Z 424.266,A -85,B 0,C 180,E1 -6229.452,E2 -6229.452} C_VEL
LIN {X 0,Y 499.811,Z 412.726,A -85,B 0,C 180,E1 -6229.759,E2 -6229.759} C_VEL
LIN {X 0,Y 497.687,Z 400.393,A -85,B 0,C 180,E1 -6230.082,E2 -6230.082} C_VEL
LIN {X 0,Y 496.697,Z 392.323,A -85,B 0,C 180,E1 -6230.254,E2 -6230.254} C_VEL
LIN {X 0,Y 497.158,Z 374.218,A -85,B 0,C 180,E1 -6233.24,E2 -6233.24} C_VEL
LIN {X 0,Y 497.83,Z 355.951,A -85,B 0,C 180,E1 -6236.404,E2 -6236.404} C_VEL
LIN {X 0,Y 498.711,Z 340.554,A -85,B 0,C 180,E1 -6239.264,E2 -6239.264} C_VEL
LIN {X 0,Y 499.841,Z 326.867,A -85,B 0,C 180,E1 -6242.059,E2 -6242.059} C_VEL
LIN {X 0,Y 501.347,Z 315.753,A -85,B 0,C 180,E1 -6244.592,E2 -6244.592} C_VEL
LIN {X 0,Y 501.602,Z 312.348,A -85,B 0,C 180,E1 -6245.477,E2 -6245.477} C_VEL
LIN {X 0,Y 500.308,Z 307.167,A -85,B 0,C 180,E1 -6247.16,E2 -6247.16} C_VEL
LIN {X 0,Y 498.888,Z 301.658,A -85,B 0,C 180,E1 -6249.341,E2 -6249.341} C_VEL
LIN {X 0,Y 497.806,Z 297.517,A -85,B 0,C 180,E1 -6251.571,E2 -6251.571} C_VEL
LIN {X 0,Y 497.214,Z 295.314,A -85,B 0,C 180,E1 -6253.286,E2 -6253.286} C_VEL
LIN {X 0,Y 496.852,Z 293.909,A -85,B 0,C 180,E1 -6255.012,E2 -6255.012} C_VEL
LIN {X 0,Y 496.582,Z 293.102,A -85,B 0,C 180,E1 -6257.387,E2 -6257.387} C_VEL
LIN {X 0,Y 496.563,Z 293.369,A -85,B 0,C 180,E1 -6259.843,E2 -6259.843} C_VEL
LIN {X 0,Y 496.668,Z 294.507,A -85,B 0,C 180,E1 -6262.522,E2 -6262.522} C_VEL
LIN {X 0,Y 496.668,Z 296.13,A -85,B 0,C 180,E1 -6265.157,E2 -6265.157} C_VEL
LIN {X 0,Y 496.495,Z 297.788,A -85,B 0,C 180,E1 -6267.459,E2 -6267.459} C_VEL
LIN {X 0,Y 496.319,Z 299.929,A -85,B 0,C 180,E1 -6270.29,E2 -6270.29} C_VEL
LIN {X 0,Y 496.226,Z 302.149,A -85,B 0,C 180,E1 -6273.16,E2 -6273.16} C_VEL
LIN {X 0,Y 496.103,Z 304.169,A -85,B 0,C 180,E1 -6275.743,E2 -6275.743} C_VEL
LIN {X 0,Y 495.986,Z 306.312,A -85,B 0,C 180,E1 -6278.382,E2 -6278.382} C_VEL
LIN {X 0,Y 495.873,Z 308.448,A -85,B 0,C 180,E1 -6280.975,E2 -6280.975} C_VEL
LIN {X 0,Y 495.771,Z 310.633,A -85,B 0,C 180,E1 -6283.53,E2 -6283.53} C_VEL
LIN {X 0,Y 495.771,Z 312.368,A -85,B 0,C 180,E1 -6285.322,E2 -6285.322} C_VEL
LIN {X 0,Y 498.769,Z 321.266,A -85,B 0,C 180,E1 -6285.724,E2 -6285.724} C_VEL
LIN {X 0,Y 498.484,Z 333.922,A -85,B 0,C 180,E1 -6286.237,E2 -6286.237} C_VEL
LIN {X 0,Y 498.13,Z 345.355,A -85,B 0,C 180,E1 -6286.855,E2 -6286.855} C_VEL
LIN {X 0,Y 497.676,Z 357.433,A -85,B 0,C 180,E1 -6287.688,E2 -6287.688} C_VEL
LIN {X 0,Y 497.294,Z 367.829,A -85,B 0,C 180,E1 -6288.589,E2 -6288.589} C_VEL
LIN {X 0,Y 496.92,Z 377.381,A -85,B 0,C 180,E1 -6289.611,E2 -6289.611} C_VEL
LIN {X 0,Y 496.52,Z 386.683,A -85,B 0,C 180,E1 -6290.837,E2 -6290.837} C_VEL
LIN {X 0,Y 496.189,Z 394.245,A -85,B 0,C 180,E1 -6292.083,E2 -6292.083} C_VEL
LIN {X 0,Y 495.98,Z 400.952,A -85,B 0,C 180,E1 -6293.491,E2 -6293.491} C_VEL
LIN {X 0,Y 495.724,Z 405.506,A -85,B 0,C 180,E1 -6294.713,E2 -6294.713} C_VEL
LIN {X 0,Y 495.591,Z 408.967,A -85,B 0,C 180,E1 -6295.934,E2 -6295.934} C_VEL
LIN {X 0,Y 495.642,Z 410.718,A -85,B 0,C 180,E1 -6296.749,E2 -6296.749} C_VEL
LIN {X 0,Y 495.494,Z 412.066,A -85,B 0,C 180,E1 -6297.561,E2 -6297.561} C_VEL
LIN {X 0,Y 495.371,Z 412.995,A -85,B 0,C 180,E1 -6298.374,E2 -6298.374} C_VEL
LIN {X 0,Y 495.427,Z 413.515,A -85,B 0,C 180,E1 -6299.187,E2 -6299.187} C_VEL
LIN {X 0,Y 495.413,Z 413.67,A -85,B 0,C 180,E1 -6300,E2 -6300} C_VEL
LIN {X 0,Y 495.412,Z 413.42,A -85,B 0,C 180,E1 -6300.813,E2 -6300.813} C_VEL
LIN {X 0,Y 495.344,Z 411.735,A -85,B 0,C 180,E1 -6302.44,E2 -6302.44} C_VEL
LIN {X 0,Y 495.417,Z 410.295,A -85,B 0,C 180,E1 -6303.253,E2 -6303.253} C_VEL
LIN {X 0,Y 495.548,Z 407.313,A -85,B 0,C 180,E1 -6304.474,E2 -6304.474} C_VEL
LIN {X 0,Y 495.572,Z 403.336,A -85,B 0,C 180,E1 -6305.697,E2 -6305.697} C_VEL
LIN {X 0,Y 495.772,Z 398.838,A -85,B 0,C 180,E1 -6306.783,E2 -6306.783} C_VEL
LIN {X 0,Y 495.966,Z 391.813,A -85,B 0,C 180,E1 -6308.147,E2 -6308.147} C_VEL
LIN {X 0,Y 496.259,Z 383.823,A -85,B 0,C 180,E1 -6309.373,E2 -6309.373} C_VEL
LIN {X 0,Y 496.518,Z 375.709,A -85,B 0,C 180,E1 -6310.397,E2 -6310.397} C_VEL
LIN {X 0,Y 496.953,Z 365.829,A -85,B 0,C 180,E1 -6311.42,E2 -6311.42} C_VEL
LIN {X 0,Y 497.228,Z 356.204,A -85,B 0,C 180,E1 -6312.241,E2 -6312.241} C_VEL
LIN {X 0,Y 497.622,Z 344.214,A -85,B 0,C 180,E1 -6313.06,E2 -6313.06} C_VEL
LIN {X 0,Y 497.941,Z 331.588,A -85,B 0,C 180,E1 -6313.727,E2 -6313.727} C_VEL
LIN {X 0,Y 498.023,Z 319.476,A -85,B 0,C 180,E1 -6314.21,E2 -6314.21} C_VEL
LIN {X 0,Y 495.25,Z 308.358,A -85,B 0,C 180,E1 -6314.642,E2 -6314.642} C_VEL
LIN {X 0,Y 495.234,Z 304.482,A -85,B 0,C 180,E1 -6318.192,E2 -6318.192} C_VEL
LIN {X 0,Y 495.268,Z 301.69,A -85,B 0,C 180,E1 -6320.779,E2 -6320.779} C_VEL
LIN {X 0,Y 495.248,Z 298.894,A -85,B 0,C 180,E1 -6323.412,E2 -6323.412} C_VEL
LIN {X 0,Y 495.281,Z 296.007,A -85,B 0,C 180,E1 -6326.097,E2 -6326.097} C_VEL
LIN {X 0,Y 495.354,Z 293.079,A -85,B 0,C 180,E1 -6328.841,E2 -6328.841} C_VEL
LIN {X 0,Y 495.347,Z 290.069,A -85,B 0,C 180,E1 -6331.665,E2 -6331.665} C_VEL
LIN {X 0,Y 495.349,Z 289.411,A -85,B 0,C 180,E1 -6332.625,E2 -6332.625} C_VEL
LIN {X 0,Y 495.668,Z 289.37,A -85,B 0,C 180,E1 -6335.544,E2 -6335.544} C_VEL
LIN {X 0,Y 495.767,Z 289.357,A -85,B 0,C 180,E1 -6338.768,E2 -6338.768} C_VEL
LIN {X 0,Y 495.759,Z 289.352,A -85,B 0,C 180,E1 -6341.781,E2 -6341.781} C_VEL
LIN {X 0,Y 495.739,Z 289.356,A -85,B 0,C 180,E1 -6345.141,E2 -6345.141} C_VEL
LIN {X 0,Y 495.712,Z 289.366,A -85,B 0,C 180,E1 -6348.214,E2 -6348.214} C_VEL
LIN {X 0,Y 495.671,Z 289.37,A -85,B 0,C 180,E1 -6349.29,E2 -6349.29} C_VEL
LIN {X 0,Y 495.692,Z 290.652,A -85,B 0,C 180,E1 -6350.356,E2 -6350.356} C_VEL
LIN {X 0,Y 495.647,Z 295.229,A -85,B 0,C 180,E1 -6353.449,E2 -6353.449} C_VEL
LIN {X 0,Y 495.598,Z 299.341,A -85,B 0,C 180,E1 -6356.423,E2 -6356.423} C_VEL
LIN {X 0,Y 495.595,Z 299.681,A -85,B 0,C 180,E1 -6356.676,E2 -6356.676} C_VEL
LIN {X 0,Y 494.932,Z 300.673,A -85,B 0,C 180,E1 -6357.344,E2 -6357.344} C_VEL
LIN {X 0,Y 492.052,Z 302.519,A -85,B 0,C 180,E1 -6358.424,E2 -6358.424} C_VEL
LIN {X 0,Y 489.602,Z 304.019,A -85,B 0,C 180,E1 -6359.295,E2 -6359.295} C_VEL
LIN {X 0,Y 488.539,Z 305.042,A -85,B 0,C 180,E1 -6359.969,E2 -6359.969} C_VEL
LIN {X 0,Y 488.447,Z 305.354,A -85,B 0,C 180,E1 -6360.198,E2 -6360.198} C_VEL
LIN {X 0,Y 488.424,Z 309.355,A -85,B 0,C 180,E1 -6363.142,E2 -6363.142} C_VEL
LIN {X 0,Y 488.346,Z 313.787,A -85,B 0,C 180,E1 -6366.236,E2 -6366.236} C_VEL
LIN {X 0,Y 488.404,Z 318.642,A -85,B 0,C 180,E1 -6369.282,E2 -6369.282} C_VEL
LIN {X 0,Y 493.42,Z 334.242,A -85,B 0,C 180,E1 -6369.838,E2 -6369.838} C_VEL
LIN {X 0,Y 494.1,Z 338.096,A -85,B 0,C 180,E1 -6369.976,E2 -6369.976} C_VEL
LIN {X 0,Y 493.744,Z 352.241,A -85,B 0,C 180,E1 -6370.46,E2 -6370.46} C_VEL
LIN {X 0,Y 493.127,Z 366.026,A -85,B 0,C 180,E1 -6371.081,E2 -6371.081} C_VEL
LIN {X 0,Y 492.567,Z 380.387,A -85,B 0,C 180,E1 -6371.921,E2 -6371.921} C_VEL
LIN {X 0,Y 491.858,Z 393.387,A -85,B 0,C 180,E1 -6372.86,E2 -6372.86} C_VEL
LIN {X 0,Y 491.209,Z 404.945,A -85,B 0,C 180,E1 -6373.872,E2 -6373.872} C_VEL
LIN {X 0,Y 490.547,Z 416.284,A -85,B 0,C 180,E1 -6375.055,E2 -6375.055} C_VEL
LIN {X 0,Y 489.964,Z 426.38,A -85,B 0,C 180,E1 -6376.309,E2 -6376.309} C_VEL
LIN {X 0,Y 489.341,Z 436.357,A -85,B 0,C 180,E1 -6377.787,E2 -6377.787} C_VEL
LIN {X 0,Y 488.912,Z 444.427,A -85,B 0,C 180,E1 -6379.23,E2 -6379.23} C_VEL
LIN {X 0,Y 488.538,Z 452.083,A -85,B 0,C 180,E1 -6380.895,E2 -6380.895} C_VEL
LIN {X 0,Y 488.3,Z 458.166,A -85,B 0,C 180,E1 -6382.557,E2 -6382.557} C_VEL
LIN {X 0,Y 488.15,Z 462.868,A -85,B 0,C 180,E1 -6384.216,E2 -6384.216} C_VEL
LIN {X 0,Y 488.052,Z 466.318,A -85,B 0,C 180,E1 -6385.871,E2 -6385.871} C_VEL
LIN {X 0,Y 487.994,Z 468.595,A -85,B 0,C 180,E1 -6387.524,E2 -6387.524} C_VEL
LIN {X 0,Y 487.871,Z 469.763,A -85,B 0,C 180,E1 -6389.174,E2 -6389.174} C_VEL
LIN {X 0,Y 487.871,Z 469.779,A -85,B 0,C 180,E1 -6390.825,E2 -6390.825} C_VEL
LIN {X 0,Y 487.994,Z 468.675,A -85,B 0,C 180,E1 -6392.476,E2 -6392.476} C_VEL
LIN {X 0,Y 488.052,Z 466.466,A -85,B 0,C 180,E1 -6394.129,E2 -6394.129} C_VEL
LIN {X 0,Y 488.146,Z 463.093,A -85,B 0,C 180,E1 -6395.784,E2 -6395.784} C_VEL
LIN {X 0,Y 488.299,Z 458.467,A -85,B 0,C 180,E1 -6397.443,E2 -6397.443} C_VEL
LIN {X 0,Y 488.518,Z 452.458,A -85,B 0,C 180,E1 -6399.105,E2 -6399.105} C_VEL
LIN {X 0,Y 488.897,Z 444.887,A -85,B 0,C 180,E1 -6400.77,E2 -6400.77} C_VEL
LIN {X 0,Y 489.309,Z 437.105,A -85,B 0,C 180,E1 -6402.183,E2 -6402.183} C_VEL
LIN {X 0,Y 489.81,Z 428.574,A -85,B 0,C 180,E1 -6403.483,E2 -6403.483} C_VEL
LIN {X 0,Y 490.386,Z 418.84,A -85,B 0,C 180,E1 -6404.737,E2 -6404.737} C_VEL
LIN {X 0,Y 491.045,Z 407.726,A -85,B 0,C 180,E1 -6405.945,E2 -6405.945} C_VEL
LIN {X 0,Y 491.726,Z 396.197,A -85,B 0,C 180,E1 -6406.994,E2 -6406.994} C_VEL
LIN {X 0,Y 492.404,Z 383.192,A -85,B 0,C 180,E1 -6407.978,E2 -6407.978} C_VEL
LIN {X 0,Y 492.99,Z 369.555,A -85,B 0,C 180,E1 -6408.816,E2 -6408.816} C_VEL
LIN {X 0,Y 493.645,Z 355.066,A -85,B 0,C 180,E1 -6409.512,E2 -6409.512} C_VEL
LIN {X 0,Y 494.029,Z 340.535,A -85,B 0,C 180,E1 -6410.04,E2 -6410.04} C_VEL
LIN {X 0,Y 493.975,Z 336.473,A -85,B 0,C 180,E1 -6410.169,E2 -6410.169} C_VEL
LIN {X 0,Y 490.051,Z 323.546,A -85,B 0,C 180,E1 -6410.648,E2 -6410.648} C_VEL
LIN {X 0,Y 488.363,Z 318.464,A -85,B 0,C 180,E1 -6410.824,E2 -6410.824} C_VEL
LIN {X 0,Y 488.344,Z 313.936,A -85,B 0,C 180,E1 -6413.763,E2 -6413.763} C_VEL
LIN {X 0,Y 488.431,Z 309.476,A -85,B 0,C 180,E1 -6416.86,E2 -6416.86} C_VEL
LIN {X 0,Y 488.452,Z 306.152,A -85,B 0,C 180,E1 -6419.288,E2 -6419.288} C_VEL
LIN {X 0,Y 488.541,Z 302.325,A -85,B 0,C 180,E1 -6422.159,E2 -6422.159} C_VEL
LIN {X 0,Y 488.584,Z 298.308,A -85,B 0,C 180,E1 -6425.126,E2 -6425.126} C_VEL
LIN {X 0,Y 488.67,Z 293.939,A -85,B 0,C 180,E1 -6428.201,E2 -6428.201} C_VEL
LIN {X 0,Y 488.578,Z 290.331,A -85,B 0,C 180,E1 -6430.61,E2 -6430.61} C_VEL
LIN {X 0,Y 488.679,Z 290.242,A -85,B 0,C 180,E1 -6433.655,E2 -6433.655} C_VEL
LIN {X 0,Y 488.687,Z 290.238,A -85,B 0,C 180,E1 -6436.345,E2 -6436.345} C_VEL
LIN {X 0,Y 488.734,Z 290.231,A -85,B 0,C 180,E1 -6439.676,E2 -6439.676} C_VEL
LIN {X 0,Y 488.678,Z 290.237,A -85,B 0,C 180,E1 -6442.841,E2 -6442.841} C_VEL
LIN {X 0,Y 488.733,Z 290.228,A -85,B 0,C 180,E1 -6445.887,E2 -6445.887} C_VEL
LIN {X 0,Y 488.69,Z 290.236,A -85,B 0,C 180,E1 -6448.82,E2 -6448.82} C_VEL
LIN {X 0,Y 488.691,Z 290.237,A -85,B 0,C 180,E1 -6451.668,E2 -6451.668} C_VEL
LIN {X 0,Y 488.703,Z 290.232,A -85,B 0,C 180,E1 -6454.958,E2 -6454.958} C_VEL
LIN {X 0,Y 488.699,Z 290.23,A -85,B 0,C 180,E1 -6458.043,E2 -6458.043} C_VEL
LIN {X 0,Y 488.736,Z 290.231,A -85,B 0,C 180,E1 -6460.686,E2 -6460.686} C_VEL
LIN {X 0,Y 488.757,Z 290.225,A -85,B 0,C 180,E1 -6464.145,E2 -6464.145} C_VEL
LIN {X 0,Y 488.734,Z 290.233,A -85,B 0,C 180,E1 -6466.698,E2 -6466.698} C_VEL
LIN {X 0,Y 488.736,Z 290.226,A -85,B 0,C 180,E1 -6469.226,E2 -6469.226} C_VEL
LIN {X 0,Y 488.771,Z 290.229,A -85,B 0,C 180,E1 -6471.733,E2 -6471.733} C_VEL
LIN {X 0,Y 488.826,Z 290.212,A -85,B 0,C 180,E1 -6474.224,E2 -6474.224} C_VEL
LIN {X 0,Y 488.96,Z 290.201,A -85,B 0,C 180,E1 -6477.529,E2 -6477.529} C_VEL
LIN {X 0,Y 488.971,Z 290.194,A -85,B 0,C 180,E1 -6480,E2 -6480} C_VEL
LIN {X 0,Y 488.952,Z 290.203,A -85,B 0,C 180,E1 -6482.471,E2 -6482.471} C_VEL
LIN {X 0,Y 488.822,Z 290.214,A -85,B 0,C 180,E1 -6485.776,E2 -6485.776} C_VEL
LIN {X 0,Y 488.787,Z 290.225,A -85,B 0,C 180,E1 -6488.267,E2 -6488.267} C_VEL
LIN {X 0,Y 488.806,Z 290.214,A -85,B 0,C 180,E1 -6491.612,E2 -6491.612} C_VEL
LIN {X 0,Y 488.753,Z 290.23,A -85,B 0,C 180,E1 -6495.001,E2 -6495.001} C_VEL
LIN {X 0,Y 488.747,Z 290.23,A -85,B 0,C 180,E1 -6498.442,E2 -6498.442} C_VEL
LIN {X 0,Y 488.707,Z 290.228,A -85,B 0,C 180,E1 -6501.071,E2 -6501.071} C_VEL
LIN {X 0,Y 488.67,Z 290.242,A -85,B 0,C 180,E1 -6503.747,E2 -6503.747} C_VEL
LIN {X 0,Y 488.7,Z 290.232,A -85,B 0,C 180,E1 -6506.922,E2 -6506.922} C_VEL
LIN {X 0,Y 488.724,Z 290.236,A -85,B 0,C 180,E1 -6510.219,E2 -6510.219} C_VEL
LIN {X 0,Y 488.734,Z 290.234,A -85,B 0,C 180,E1 -6513.484,E2 -6513.484} C_VEL
LIN {X 0,Y 488.672,Z 290.238,A -85,B 0,C 180,E1 -6516.353,E2 -6516.353} C_VEL
LIN {X 0,Y 488.696,Z 290.235,A -85,B 0,C 180,E1 -6519.255,E2 -6519.255} C_VEL
LIN {X 0,Y 488.707,Z 290.235,A -85,B 0,C 180,E1 -6521.6,E2 -6521.6} C_VEL
LIN {X 0,Y 488.7,Z 290.233,A -85,B 0,C 180,E1 -6524.803,E2 -6524.803} C_VEL
LIN {X 0,Y 488.666,Z 290.236,A -85,B 0,C 180,E1 -6527.472,E2 -6527.472} C_VEL
LIN {X 0,Y 488.716,Z 290.337,A -85,B 0,C 180,E1 -6529.065,E2 -6529.065} C_VEL
LIN {X 0,Y 491.84,Z 302.488,A -85,B 0,C 180,E1 -6532.089,E2 -6532.089} C_VEL
LIN {X 0,Y 494.461,Z 313.292,A -85,B 0,C 180,E1 -6534.606,E2 -6534.606} C_VEL
LIN {X 0,Y 493.654,Z 324.084,A -85,B 0,C 180,E1 -6536.763,E2 -6536.763} C_VEL
LIN {X 0,Y 492.593,Z 338.627,A -85,B 0,C 180,E1 -6539.57,E2 -6539.57} C_VEL
LIN {X 0,Y 491.632,Z 353.818,A -85,B 0,C 180,E1 -6542.412,E2 -6542.412} C_VEL
LIN {X 0,Y 490.71,Z 371.943,A -85,B 0,C 180,E1 -6545.685,E2 -6545.685} C_VEL
LIN {X 0,Y 489.929,Z 392.049,A -85,B 0,C 180,E1 -6549.204,E2 -6549.204} C_VEL
LIN {X 0,Y 489.873,Z 393.43,A -85,B 0,C 180,E1 -6549.445,E2 -6549.445} C_VEL
LIN {X 0,Y 492.457,Z 410.042,A -85,B 0,C 180,E1 -6549.842,E2 -6549.842} C_VEL
LIN {X 0,Y 493.272,Z 414.474,A -85,B 0,C 180,E1 -6549.978,E2 -6549.978} C_VEL
LIN {X 0,Y 492.786,Z 429.512,A -85,B 0,C 180,E1 -6550.434,E2 -6550.434} C_VEL
LIN {X 0,Y 492.249,Z 444.246,A -85,B 0,C 180,E1 -6551.046,E2 -6551.046} C_VEL
LIN {X 0,Y 491.635,Z 457.934,A -85,B 0,C 180,E1 -6551.778,E2 -6551.778} C_VEL
LIN {X 0,Y 490.99,Z 472.097,A -85,B 0,C 180,E1 -6552.722,E2 -6552.722} C_VEL
LIN {X 0,Y 490.386,Z 485.138,A -85,B 0,C 180,E1 -6553.783,E2 -6553.783} C_VEL
